(* CODESYS project SWDM240HES_S00107_20240509.project
   Company: ifm electronic
   Description: CR721S 2.25MByte Standard and Safety
   Title: ifmCR721S_TemplateProject
   Version: 3.1.4.1

Project tree, tasks and I/O mapping:
  StandardPLC : CR721S Standard, ifm electronic, order no. CR721S, version 3.1.4.1
    application Application
      libraries: ifmR360-3, * (ifm electronic); Standard, * (System); Util, * (System); SWMC_C_LIB, 3.5.15.7 (SW); CoDeSys External Library Template, 3.5.16.40 (3S - Smart Software Solutions GmbH); CoDeSys Common Library Template, 3.5.11.0 (3S - Smart Software Solutions GmbH)
      task Task (cyclic, interval t#10ms, priority 0) calls PLC_PRG
      IO_CONFIG/
        function block DiagFunction [FBD]
        program OUTPUT_CONFID [FBD]
        program ConfigDiagProt [FBD]
        program INPUT_CONFIG_PI [FBD]
        program INPUT_CONFIG [ST]
      EVC
      program PLC_PRG [FBD]
      CAN/
        program CAN1 [ST]
        program GPS_TONGXING_ALL [ST]
        program GPS_ALL [ST]
        program CanRecover [ST]
        program CAN0 [ST]
        program CAN2 [ST]
        program CAN_J [ST]
      data type FIFO_DUT
      SaveEngine/
        program SaveEngine [ST]
        global variables GVL_SaveEngine
        program SaveEngineControl [ST]
        program SaveEngineMode_1 [ST]
        program SaveEngineMode_2 [ST]
        program SaveEngineMode_3 [ST]
        program SaveEngineMode_4 [ST]
        program SaveEngineMode_5 [ST]
        program SaveEngineMode_6 [ST]
        program SaveEngineMode_7 [ST]
        program SaveEngineMode_8 [ST]
        program SaveEngineMode_19 [ST]
        program SaveEngineMode_10 [ST]
        program SaveEngineMode_11 [ST]
        program SaveEngineMode_12 [ST]
        program SaveEngineMode_9 [ST]
        program MainWinTension_Ave [ST]
        program Wt_Cal [ST]
      MOVE/
        program MastControl [ST]
        program worktime [ST]
        function block PID_JYF [ST]
        function block curve_quxian [ST]
        program control [ST]
        program inti_fasle [ST]
        program Joy_Analog_output [ST]
        function block ROTATE_AUTO [ST]
        function block MODE_ROTATE [ST]
      CAIJI/
        function block PRESSURE [ST]
        function block ANGLE_CAIJI_Y [ST]
        function block DEPTH [ST]
        function block Tension [ST]
        function block ZONGXIANJISUAN [ST]
        function block CAN_XY [FBD]
        function block censor_cali [FBD]
        function block FUEL_LEVEL [ST]
        function block ANGLE_CAIJI_X [ST]
        function block HYD_OIL_TEM [ST]
        program CAIJI_DEPTH [ST]
      GLV/
        global variables PersistentVars
        global variables Global_Variablen
        global variables IO_GLV
        global variables CAN_GVL
    HMI : HMI, ifm electronic, version 3.1.4.1
      User_LEDs : User_LEDs, ifm electronic, version 3.1.4.1
          input  UserLED0_I : LED_IEC_B_INPUT_MAPPING_TYPE  // UserLED0_I
          input  UserLED1_I : LED_IEC_B_INPUT_MAPPING_TYPE  // UserLED1_I
          input  UserLED2_I : LED_IEC_B_INPUT_MAPPING_TYPE  // UserLED2_I
          input  UserLED3_I : LED_IEC_B_INPUT_MAPPING_TYPE  // UserLED3_I
          output UserLED0_Q : LED_IEC_B_OUTPUT_MAPPING_TYPE  // User LED 0
          output UserLED1_Q : LED_IEC_B_OUTPUT_MAPPING_TYPE  // User LED 1
          output UserLED2_Q : LED_IEC_B_OUTPUT_MAPPING_TYPE  // User LED 2
          output UserLED3_Q : LED_IEC_B_OUTPUT_MAPPING_TYPE  // User LED 3
    Local_IO : Local_IO, ifm electronic, version 3.1.4.1
      System_Inputs : System_Inputs, ifm electronic, version 3.1.4.1
          input  VBB30 : IN_SYSTEM_VOLTAGE_INPUT_MAPPING_TYPE  // VBB30
          input  VBB15 : IN_SYSTEM_VOLTAGE_INPUT_MAPPING_TYPE  // VBB15
          input  TemperatureBoard0 : IN_TEMPERATURE_INPUT_MAPPING_TYPE  // TemperatureBoard0
          input  TemperatureChip0 : IN_TEMPERATURE_INPUT_MAPPING_TYPE  // TemperatureChip0
      Inputs : Inputs, ifm electronic, version 3.1.4.1
          input  IN0100_I : IN_MULTIFUNCTION_A_INPUT_MAPPING_TYPE  // IN0100_I
          input  IN0101_I : IN_MULTIFUNCTION_A_INPUT_MAPPING_TYPE  // IN0101_I
          input  IN0102_I : IN_MULTIFUNCTION_A_INPUT_MAPPING_TYPE  // IN0102_I
          input  IN0103_I : IN_MULTIFUNCTION_A_INPUT_MAPPING_TYPE  // IN0103_I
          input  IN0200_I : IN_MULTIFUNCTION_A_INPUT_MAPPING_TYPE  // IN0200_I
          input  IN0201_I : IN_MULTIFUNCTION_A_INPUT_MAPPING_TYPE  // IN0201_I
          input  IN0202_I : IN_MULTIFUNCTION_A_INPUT_MAPPING_TYPE  // IN0202_I
          input  IN0203_I : IN_MULTIFUNCTION_A_INPUT_MAPPING_TYPE  // IN0203_I
          input  IN0600_I : IN_MULTIFUNCTION_A_INPUT_MAPPING_TYPE  // IN0600_I
          input  IN0601_I : IN_MULTIFUNCTION_A_INPUT_MAPPING_TYPE  // IN0601_I
          input  IN0602_I : IN_MULTIFUNCTION_A_INPUT_MAPPING_TYPE  // IN0602_I
          input  IN0603_I : IN_MULTIFUNCTION_A_INPUT_MAPPING_TYPE  // IN0603_I
          input  IN0700_I : IN_MULTIFUNCTION_A_INPUT_MAPPING_TYPE  // IN0700_I
          input  IN0701_I : IN_MULTIFUNCTION_A_INPUT_MAPPING_TYPE  // IN0701_I
          input  IN0702_I : IN_MULTIFUNCTION_A_INPUT_MAPPING_TYPE  // IN0702_I
          input  IN0703_I : IN_MULTIFUNCTION_A_INPUT_MAPPING_TYPE  // IN0703_I
          input  IN1100_I : IN_MULTIFUNCTION_A_INPUT_MAPPING_TYPE  // IN1100_I
          input  IN1101_I : IN_MULTIFUNCTION_A_INPUT_MAPPING_TYPE  // IN1101_I
          input  IN1102_I : IN_MULTIFUNCTION_A_INPUT_MAPPING_TYPE  // IN1102_I
          input  IN1103_I : IN_MULTIFUNCTION_A_INPUT_MAPPING_TYPE  // IN1103_I
          input  IN1600_I : IN_MULTIFUNCTION_A_INPUT_MAPPING_TYPE  // IN1600_I
          input  IN1601_I : IN_MULTIFUNCTION_A_INPUT_MAPPING_TYPE  // IN1601_I
          input  IN1602_I : IN_MULTIFUNCTION_A_INPUT_MAPPING_TYPE  // IN1602_I
          input  IN1603_I : IN_MULTIFUNCTION_A_INPUT_MAPPING_TYPE  // IN1603_I
          input  IN0400_I : IN_RESISTOR_A_INPUT_MAPPING_TYPE  // IN0400_I
          input  IN0401_I : IN_RESISTOR_A_INPUT_MAPPING_TYPE  // IN0401_I
          input  IN0900_I : IN_RESISTOR_A_INPUT_MAPPING_TYPE  // IN0900_I
          input  IN0901_I : IN_RESISTOR_A_INPUT_MAPPING_TYPE  // IN0901_I
          input  IN1200_I : IN_DIGITAL_A_INPUT_MAPPING_TYPE  // IN1200_I
          input  IN1201_I : IN_DIGITAL_A_INPUT_MAPPING_TYPE  // IN1201_I
          input  IN1202_I : IN_DIGITAL_A_INPUT_MAPPING_TYPE  // IN1202_I
          input  IN1203_I : IN_DIGITAL_A_INPUT_MAPPING_TYPE  // IN1203_I
          input  IN1400_I : IN_DIGITAL_A_INPUT_MAPPING_TYPE  // IN1400_I
          input  IN1401_I : IN_DIGITAL_A_INPUT_MAPPING_TYPE  // IN1401_I
          input  IN1402_I : IN_DIGITAL_A_INPUT_MAPPING_TYPE  // IN1402_I
          input  IN1403_I : IN_DIGITAL_A_INPUT_MAPPING_TYPE  // IN1403_I
          input  IN1700_I : IN_DIGITAL_A_INPUT_MAPPING_TYPE  // IN1700_I
          input  IN1701_I : IN_DIGITAL_A_INPUT_MAPPING_TYPE  // IN1701_I
          input  IN1702_I : IN_DIGITAL_A_INPUT_MAPPING_TYPE  // IN1702_I
          input  IN1703_I : IN_DIGITAL_A_INPUT_MAPPING_TYPE  // IN1703_I
          input  IN1800_I : IN_DIGITAL_A_INPUT_MAPPING_TYPE  // IN1800_I
          input  IN1801_I : IN_DIGITAL_A_INPUT_MAPPING_TYPE  // IN1801_I
          input  IN1802_I : IN_DIGITAL_A_INPUT_MAPPING_TYPE  // IN1802_I
          input  IN1803_I : IN_DIGITAL_A_INPUT_MAPPING_TYPE  // IN1803_I
          input  IN0300_I : IN_DIGITAL_B_INPUT_MAPPING_TYPE  // IN0300_I
          input  IN0301_I : IN_DIGITAL_B_INPUT_MAPPING_TYPE  // IN0301_I
          input  IN0800_I : IN_DIGITAL_B_INPUT_MAPPING_TYPE  // IN0800_I
          input  IN0801_I : IN_DIGITAL_B_INPUT_MAPPING_TYPE  // IN0801_I
          input  IN1300_I : IN_DIGITAL_B_INPUT_MAPPING_TYPE  // IN1300_I
          input  IN1301_I : IN_DIGITAL_B_INPUT_MAPPING_TYPE  // IN1301_I
          input  IN1302_I : IN_DIGITAL_B_INPUT_MAPPING_TYPE  // IN1302_I
          input  IN1303_I : IN_DIGITAL_B_INPUT_MAPPING_TYPE  // IN1303_I
          input  COM_RESET_I : IN_COMMUNICATION_RESET_INPUT_MAPPING_TYPE  // COM_RESET_I
          input  IN0000_I : IN_FREQUENCY_B_CHANNEL_A_INPUT_MAPPING_TYPE  // IN0000_I
          input  IN0002_I : IN_FREQUENCY_B_CHANNEL_A_INPUT_MAPPING_TYPE  // IN0002_I
          input  IN0500_I : IN_FREQUENCY_B_CHANNEL_A_INPUT_MAPPING_TYPE  // IN0500_I
          input  IN0502_I : IN_FREQUENCY_B_CHANNEL_A_INPUT_MAPPING_TYPE  // IN0502_I
          input  IN1000_I : IN_FREQUENCY_B_CHANNEL_A_INPUT_MAPPING_TYPE  // IN1000_I
          input  IN1002_I : IN_FREQUENCY_B_CHANNEL_A_INPUT_MAPPING_TYPE  // IN1002_I
          input  IN1500_I : IN_FREQUENCY_B_CHANNEL_A_INPUT_MAPPING_TYPE  // IN1500_I
          input  IN1502_I : IN_FREQUENCY_B_CHANNEL_A_INPUT_MAPPING_TYPE  // IN1502_I
          input  IN0001_I : IN_FREQUENCY_B_CHANNEL_B_INPUT_MAPPING_TYPE  // IN0001_I
          input  IN0003_I : IN_FREQUENCY_B_CHANNEL_B_INPUT_MAPPING_TYPE  // IN0003_I
          input  IN0501_I : IN_FREQUENCY_B_CHANNEL_B_INPUT_MAPPING_TYPE  // IN0501_I
          input  IN0503_I : IN_FREQUENCY_B_CHANNEL_B_INPUT_MAPPING_TYPE  // IN0503_I
          input  IN1001_I : IN_FREQUENCY_B_CHANNEL_B_INPUT_MAPPING_TYPE  // IN1001_I
          input  IN1003_I : IN_FREQUENCY_B_CHANNEL_B_INPUT_MAPPING_TYPE  // IN1003_I
          input  IN1501_I : IN_FREQUENCY_B_CHANNEL_B_INPUT_MAPPING_TYPE  // IN1501_I
          input  IN1503_I : IN_FREQUENCY_B_CHANNEL_B_INPUT_MAPPING_TYPE  // IN1503_I
      Outputs : Outputs, ifm electronic, version 3.1.4.1
          input  OUT0006_I : OUT_PWM_40_BRIDGE_A_INPUT_MAPPING_TYPE  // OUT0006_I
          input  OUT0106_I : OUT_PWM_40_BRIDGE_A_INPUT_MAPPING_TYPE  // OUT0106_I
          input  OUT0206_I : OUT_PWM_40_BRIDGE_A_INPUT_MAPPING_TYPE  // OUT0206_I
          input  OUT0306_I : OUT_PWM_40_BRIDGE_A_INPUT_MAPPING_TYPE  // OUT0306_I
          input  OUT0406_I : OUT_PWM_40_BRIDGE_A_INPUT_MAPPING_TYPE  // OUT0406_I
          input  OUT0506_I : OUT_PWM_40_BRIDGE_A_INPUT_MAPPING_TYPE  // OUT0506_I
          input  OUT0008_I : OUT_PWM_40_A_INPUT_MAPPING_TYPE  // OUT0008_I
          input  OUT0108_I : OUT_PWM_40_A_INPUT_MAPPING_TYPE  // OUT0108_I
          input  OUT0208_I : OUT_PWM_40_A_INPUT_MAPPING_TYPE  // OUT0208_I
          input  OUT0308_I : OUT_PWM_40_A_INPUT_MAPPING_TYPE  // OUT0308_I
          input  OUT0408_I : OUT_PWM_40_A_INPUT_MAPPING_TYPE  // OUT0408_I
          input  OUT0508_I : OUT_PWM_40_A_INPUT_MAPPING_TYPE  // OUT0508_I
          input  OUT0000_I : OUT_PWM_25_A_INPUT_MAPPING_TYPE  // OUT0000_I
          input  OUT0002_I : OUT_PWM_25_A_INPUT_MAPPING_TYPE  // OUT0002_I
          input  OUT0004_I : OUT_PWM_25_A_INPUT_MAPPING_TYPE  // OUT0004_I
          input  OUT0100_I : OUT_PWM_25_A_INPUT_MAPPING_TYPE  // OUT0100_I
          input  OUT0102_I : OUT_PWM_25_A_INPUT_MAPPING_TYPE  // OUT0102_I
          input  OUT0104_I : OUT_PWM_25_A_INPUT_MAPPING_TYPE  // OUT0104_I
          input  OUT0200_I : OUT_PWM_25_A_INPUT_MAPPING_TYPE  // OUT0200_I
          input  OUT0202_I : OUT_PWM_25_A_INPUT_MAPPING_TYPE  // OUT0202_I
          input  OUT0204_I : OUT_PWM_25_A_INPUT_MAPPING_TYPE  // OUT0204_I
          input  OUT0300_I : OUT_PWM_25_A_INPUT_MAPPING_TYPE  // OUT0300_I
          input  OUT0302_I : OUT_PWM_25_A_INPUT_MAPPING_TYPE  // OUT0302_I
          input  OUT0304_I : OUT_PWM_25_A_INPUT_MAPPING_TYPE  // OUT0304_I
          input  OUT0400_I : OUT_PWM_25_A_INPUT_MAPPING_TYPE  // OUT0400_I
          input  OUT0402_I : OUT_PWM_25_A_INPUT_MAPPING_TYPE  // OUT0402_I
          input  OUT0404_I : OUT_PWM_25_A_INPUT_MAPPING_TYPE  // OUT0404_I
          input  OUT0500_I : OUT_PWM_25_A_INPUT_MAPPING_TYPE  // OUT0500_I
          input  OUT0502_I : OUT_PWM_25_A_INPUT_MAPPING_TYPE  // OUT0502_I
          input  OUT0504_I : OUT_PWM_25_A_INPUT_MAPPING_TYPE  // OUT0504_I
          input  OUT3001_I : OUT_VOLTAGE_A_INPUT_MAPPING_TYPE  // OUT3001_I
          input  OUT3002_I : OUT_VOLTAGE_A_INPUT_MAPPING_TYPE  // OUT3002_I
          input  OUT3000_I : OUT_SUPPLY_A_INPUT_MAPPING_TYPE  // OUT3000_I
          input  OUT0001_I : OUT_PWM_25_B_INPUT_MAPPING_TYPE  // OUT0001_I
          input  OUT0003_I : OUT_PWM_25_B_INPUT_MAPPING_TYPE  // OUT0003_I
          input  OUT0005_I : OUT_PWM_25_B_INPUT_MAPPING_TYPE  // OUT0005_I
          input  OUT0101_I : OUT_PWM_25_B_INPUT_MAPPING_TYPE  // OUT0101_I
          input  OUT0103_I : OUT_PWM_25_B_INPUT_MAPPING_TYPE  // OUT0103_I
          input  OUT0105_I : OUT_PWM_25_B_INPUT_MAPPING_TYPE  // OUT0105_I
          input  OUT0201_I : OUT_PWM_25_B_INPUT_MAPPING_TYPE  // OUT0201_I
          input  OUT0203_I : OUT_PWM_25_B_INPUT_MAPPING_TYPE  // OUT0203_I
          input  OUT0205_I : OUT_PWM_25_B_INPUT_MAPPING_TYPE  // OUT0205_I
          input  OUT0301_I : OUT_PWM_25_B_INPUT_MAPPING_TYPE  // OUT0301_I
          input  OUT0303_I : OUT_PWM_25_B_INPUT_MAPPING_TYPE  // OUT0303_I
          input  OUT0305_I : OUT_PWM_25_B_INPUT_MAPPING_TYPE  // OUT0305_I
          input  OUT0401_I : OUT_PWM_25_B_INPUT_MAPPING_TYPE  // OUT0401_I
          input  OUT0403_I : OUT_PWM_25_B_INPUT_MAPPING_TYPE  // OUT0403_I
          input  OUT0405_I : OUT_PWM_25_B_INPUT_MAPPING_TYPE  // OUT0405_I
          input  OUT0501_I : OUT_PWM_25_B_INPUT_MAPPING_TYPE  // OUT0501_I
          input  OUT0503_I : OUT_PWM_25_B_INPUT_MAPPING_TYPE  // OUT0503_I
          input  OUT0505_I : OUT_PWM_25_B_INPUT_MAPPING_TYPE  // OUT0505_I
          input  OUT0007_I : OUT_PWM_40_BRIDGE_A_INPUT_MAPPING_TYPE  // OUT0007_I
          input  OUT0107_I : OUT_PWM_40_BRIDGE_A_INPUT_MAPPING_TYPE  // OUT0107_I
          input  OUT0207_I : OUT_PWM_40_BRIDGE_A_INPUT_MAPPING_TYPE  // OUT0207_I
          input  OUT0307_I : OUT_PWM_40_BRIDGE_A_INPUT_MAPPING_TYPE  // OUT0307_I
          input  OUT0407_I : OUT_PWM_40_BRIDGE_A_INPUT_MAPPING_TYPE  // OUT0407_I
          input  OUT0507_I : OUT_PWM_40_BRIDGE_A_INPUT_MAPPING_TYPE  // OUT0507_I
          output OUT0006_Q : OUT_PWM_40_BRIDGE_A_OUTPUT_MAPPING_TYPE  // OUT0006_Q
          output OUT0106_Q : OUT_PWM_40_BRIDGE_A_OUTPUT_MAPPING_TYPE  // OUT0106_Q
          output OUT0206_Q : OUT_PWM_40_BRIDGE_A_OUTPUT_MAPPING_TYPE  // OUT0206_Q
          output OUT0306_Q : OUT_PWM_40_BRIDGE_A_OUTPUT_MAPPING_TYPE  // OUT0306_Q
          output OUT0406_Q : OUT_PWM_40_BRIDGE_A_OUTPUT_MAPPING_TYPE  // OUT0406_Q
          output OUT0506_Q : OUT_PWM_40_BRIDGE_A_OUTPUT_MAPPING_TYPE  // OUT0506_Q
          output OUT0008_Q : OUT_PWM_40_A_OUTPUT_MAPPING_TYPE  // OUT0008_Q
          output OUT0108_Q : OUT_PWM_40_A_OUTPUT_MAPPING_TYPE  // OUT0108_Q
          output OUT0208_Q : OUT_PWM_40_A_OUTPUT_MAPPING_TYPE  // OUT0208_Q
          output OUT0308_Q : OUT_PWM_40_A_OUTPUT_MAPPING_TYPE  // OUT0308_Q
          output OUT0408_Q : OUT_PWM_40_A_OUTPUT_MAPPING_TYPE  // OUT0408_Q
          output OUT0508_Q : OUT_PWM_40_A_OUTPUT_MAPPING_TYPE  // OUT0508_Q
          output OUT0000_Q : OUT_PWM_25_A_OUTPUT_MAPPING_TYPE  // OUT0000_Q
          output OUT0002_Q : OUT_PWM_25_A_OUTPUT_MAPPING_TYPE  // OUT0002_Q
          output OUT0004_Q : OUT_PWM_25_A_OUTPUT_MAPPING_TYPE  // OUT0004_Q
          output OUT0100_Q : OUT_PWM_25_A_OUTPUT_MAPPING_TYPE  // OUT0100_Q
          output OUT0102_Q : OUT_PWM_25_A_OUTPUT_MAPPING_TYPE  // OUT0102_Q
          output OUT0104_Q : OUT_PWM_25_A_OUTPUT_MAPPING_TYPE  // OUT0104_Q
          output OUT0200_Q : OUT_PWM_25_A_OUTPUT_MAPPING_TYPE  // OUT0200_Q
          output OUT0202_Q : OUT_PWM_25_A_OUTPUT_MAPPING_TYPE  // OUT0202_Q
          output OUT0204_Q : OUT_PWM_25_A_OUTPUT_MAPPING_TYPE  // OUT0204_Q
          output OUT0300_Q : OUT_PWM_25_A_OUTPUT_MAPPING_TYPE  // OUT0300_Q
          output OUT0302_Q : OUT_PWM_25_A_OUTPUT_MAPPING_TYPE  // OUT0302_Q
          output OUT0304_Q : OUT_PWM_25_A_OUTPUT_MAPPING_TYPE  // OUT0304_Q
          output OUT0400_Q : OUT_PWM_25_A_OUTPUT_MAPPING_TYPE  // OUT0400_Q
          output OUT0402_Q : OUT_PWM_25_A_OUTPUT_MAPPING_TYPE  // OUT0402_Q
          output OUT0404_Q : OUT_PWM_25_A_OUTPUT_MAPPING_TYPE  // OUT0404_Q
          output OUT0500_Q : OUT_PWM_25_A_OUTPUT_MAPPING_TYPE  // OUT0500_Q
          output OUT0502_Q : OUT_PWM_25_A_OUTPUT_MAPPING_TYPE  // OUT0502_Q
          output OUT0504_Q : OUT_PWM_25_A_OUTPUT_MAPPING_TYPE  // OUT0504_Q
          output OUT3001_Q : OUT_VOLTAGE_A_OUTPUT_MAPPING_TYPE  // OUT3001_Q
          output OUT3002_Q : OUT_VOLTAGE_A_OUTPUT_MAPPING_TYPE  // OUT3002_Q
          output OUT3000_Q : OUT_SUPPLY_A_OUTPUT_MAPPING_TYPE  // OUT3000_Q
          output OUT0001_Q : OUT_PWM_25_B_OUTPUT_MAPPING_TYPE  // OUT0001_Q
          output OUT0003_Q : OUT_PWM_25_B_OUTPUT_MAPPING_TYPE  // OUT0003_Q
          output OUT0005_Q : OUT_PWM_25_B_OUTPUT_MAPPING_TYPE  // OUT0005_Q
          output OUT0101_Q : OUT_PWM_25_B_OUTPUT_MAPPING_TYPE  // OUT0101_Q
          output OUT0103_Q : OUT_PWM_25_B_OUTPUT_MAPPING_TYPE  // OUT0103_Q
          output OUT0105_Q : OUT_PWM_25_B_OUTPUT_MAPPING_TYPE  // OUT0105_Q
          output OUT0201_Q : OUT_PWM_25_B_OUTPUT_MAPPING_TYPE  // OUT0201_Q
          output OUT0203_Q : OUT_PWM_25_B_OUTPUT_MAPPING_TYPE  // OUT0203_Q
          output OUT0205_Q : OUT_PWM_25_B_OUTPUT_MAPPING_TYPE  // OUT0205_Q
          output OUT0301_Q : OUT_PWM_25_B_OUTPUT_MAPPING_TYPE  // OUT0301_Q
          output OUT0303_Q : OUT_PWM_25_B_OUTPUT_MAPPING_TYPE  // OUT0303_Q
          output OUT0305_Q : OUT_PWM_25_B_OUTPUT_MAPPING_TYPE  // OUT0305_Q
          output OUT0401_Q : OUT_PWM_25_B_OUTPUT_MAPPING_TYPE  // OUT0401_Q
          output OUT0403_Q : OUT_PWM_25_B_OUTPUT_MAPPING_TYPE  // OUT0403_Q
          output OUT0405_Q : OUT_PWM_25_B_OUTPUT_MAPPING_TYPE  // OUT0405_Q
          output OUT0501_Q : OUT_PWM_25_B_OUTPUT_MAPPING_TYPE  // OUT0501_Q
          output OUT0503_Q : OUT_PWM_25_B_OUTPUT_MAPPING_TYPE  // OUT0503_Q
          output OUT0505_Q : OUT_PWM_25_B_OUTPUT_MAPPING_TYPE  // OUT0505_Q
          output OUT0007_Q : OUT_PWM_40_BRIDGE_A_OUTPUT_MAPPING_TYPE  // OUT0007_Q
          output OUT0107_Q : OUT_PWM_40_BRIDGE_A_OUTPUT_MAPPING_TYPE  // OUT0107_Q
          output OUT0207_Q : OUT_PWM_40_BRIDGE_A_OUTPUT_MAPPING_TYPE  // OUT0207_Q
          output OUT0307_Q : OUT_PWM_40_BRIDGE_A_OUTPUT_MAPPING_TYPE  // OUT0307_Q
          output OUT0407_Q : OUT_PWM_40_BRIDGE_A_OUTPUT_MAPPING_TYPE  // OUT0407_Q
          output OUT0507_Q : OUT_PWM_40_BRIDGE_A_OUTPUT_MAPPING_TYPE  // OUT0507_Q
      System_Outputs : System_Outputs, ifm electronic, version 3.1.4.1
          input  VBB0_SW_I : OUT_GROUP_SWITCH_INPUT_MAPPING_TYPE  // VBB0_SW_I
          input  VBB1_SW_I : OUT_GROUP_SWITCH_INPUT_MAPPING_TYPE  // VBB1_SW_I
          input  VBB2_SW_I : OUT_GROUP_SWITCH_INPUT_MAPPING_TYPE  // VBB2_SW_I
          input  VBB3_SW_I : OUT_GROUP_SWITCH_INPUT_MAPPING_TYPE  // VBB3_SW_I
          input  VBB4_SW_I : OUT_GROUP_SWITCH_INPUT_MAPPING_TYPE  // VBB4_SW_I
          input  VBB5_SW_I : OUT_GROUP_SWITCH_INPUT_MAPPING_TYPE  // VBB5_SW_I
          output VBB0_SW_Q : OUT_GROUP_SWITCH_OUTPUT_MAPPING_TYPE  // VBB0_SW_Q
          output VBB1_SW_Q : OUT_GROUP_SWITCH_OUTPUT_MAPPING_TYPE  // VBB1_SW_Q
          output VBB2_SW_Q : OUT_GROUP_SWITCH_OUTPUT_MAPPING_TYPE  // VBB2_SW_Q
          output VBB3_SW_Q : OUT_GROUP_SWITCH_OUTPUT_MAPPING_TYPE  // VBB3_SW_Q
          output VBB4_SW_Q : OUT_GROUP_SWITCH_OUTPUT_MAPPING_TYPE  // VBB4_SW_Q
          output VBB5_SW_Q : OUT_GROUP_SWITCH_OUTPUT_MAPPING_TYPE  // VBB5_SW_Q
          output SUPPLY_SWITCH_Q : OUT_SYS_SWITCH_OUTPUT_MAPPING_TYPE  // SUPPLY_SWITCH_Q
    Communication : Communication, ifm electronic, version 3.1.4.1
      CAN : CAN, ifm electronic, version 3.1.4.1
        CANbus_0 : CANbus, ifm electronic, version 1.0.1.1
      Ethernet : Ethernet, ifm electronic, version 3.1.4.1
  SafetyPLC : CR721S SIL2, ifm electronic, order no. CR721S, version 3.1.4.1
    application Application
      libraries: ifmR360-3, * (ifm electronic); Standard, * (System); Util, * (System)
      global variables EVL
    HMI : HMI, ifm electronic, version 3.1.4.1
      User_LEDs : User_LEDs, ifm electronic, version 3.1.4.1
          input  UserLED0_I : LED_IEC_B_INPUT_MAPPING_TYPE  // UserLED0_I
          input  UserLED1_I : LED_IEC_B_INPUT_MAPPING_TYPE  // UserLED1_I
          input  UserLED2_I : LED_IEC_B_INPUT_MAPPING_TYPE  // UserLED2_I
          input  UserLED3_I : LED_IEC_B_INPUT_MAPPING_TYPE  // UserLED3_I
          output UserLED0_Q : LED_IEC_B_OUTPUT_MAPPING_TYPE  // User LED 0
          output UserLED1_Q : LED_IEC_B_OUTPUT_MAPPING_TYPE  // User LED 1
          output UserLED2_Q : LED_IEC_B_OUTPUT_MAPPING_TYPE  // User LED 2
          output UserLED3_Q : LED_IEC_B_OUTPUT_MAPPING_TYPE  // User LED 3
    Local_IO : Local_IO, ifm electronic, version 3.1.4.1
      System_Outputs : System_Outputs, ifm electronic, version 3.1.4.1
          input  VBB0_SW_I : OUT_GROUP_SWITCH_INPUT_MAPPING_TYPE  // VBB0_SW_I
          input  VBB1_SW_I : OUT_GROUP_SWITCH_INPUT_MAPPING_TYPE  // VBB1_SW_I
          input  VBB2_SW_I : OUT_GROUP_SWITCH_INPUT_MAPPING_TYPE  // VBB2_SW_I
          input  VBB3_SW_I : OUT_GROUP_SWITCH_INPUT_MAPPING_TYPE  // VBB3_SW_I
          input  VBB4_SW_I : OUT_GROUP_SWITCH_INPUT_MAPPING_TYPE  // VBB4_SW_I
          input  VBB5_SW_I : OUT_GROUP_SWITCH_INPUT_MAPPING_TYPE  // VBB5_SW_I
          output VBB0_SW_Q : OUT_GROUP_SWITCH_OUTPUT_MAPPING_TYPE  // VBB0_SW_Q
          output VBB1_SW_Q : OUT_GROUP_SWITCH_OUTPUT_MAPPING_TYPE  // VBB1_SW_Q
          output VBB2_SW_Q : OUT_GROUP_SWITCH_OUTPUT_MAPPING_TYPE  // VBB2_SW_Q
          output VBB3_SW_Q : OUT_GROUP_SWITCH_OUTPUT_MAPPING_TYPE  // VBB3_SW_Q
          output VBB4_SW_Q : OUT_GROUP_SWITCH_OUTPUT_MAPPING_TYPE  // VBB4_SW_Q
          output VBB5_SW_Q : OUT_GROUP_SWITCH_OUTPUT_MAPPING_TYPE  // VBB5_SW_Q
          output SUPPLY_SWITCH_Q : OUT_SYS_SWITCH_OUTPUT_MAPPING_TYPE  // SUPPLY_SWITCH_Q
      Outputs : Outputs, ifm electronic, version 3.1.4.1
          input  OUT0006_I : OUT_PWM_40_BRIDGE_A_INPUT_MAPPING_TYPE  // OUT0006_I
          input  OUT0106_I : OUT_PWM_40_BRIDGE_A_INPUT_MAPPING_TYPE  // OUT0106_I
          input  OUT0206_I : OUT_PWM_40_BRIDGE_A_INPUT_MAPPING_TYPE  // OUT0206_I
          input  OUT0306_I : OUT_PWM_40_BRIDGE_A_INPUT_MAPPING_TYPE  // OUT0306_I
          input  OUT0406_I : OUT_PWM_40_BRIDGE_A_INPUT_MAPPING_TYPE  // OUT0406_I
          input  OUT0506_I : OUT_PWM_40_BRIDGE_A_INPUT_MAPPING_TYPE  // OUT0506_I
          input  OUT0008_I : OUT_PWM_40_A_INPUT_MAPPING_TYPE  // OUT0008_I
          input  OUT0108_I : OUT_PWM_40_A_INPUT_MAPPING_TYPE  // OUT0108_I
          input  OUT0208_I : OUT_PWM_40_A_INPUT_MAPPING_TYPE  // OUT0208_I
          input  OUT0308_I : OUT_PWM_40_A_INPUT_MAPPING_TYPE  // OUT0308_I
          input  OUT0408_I : OUT_PWM_40_A_INPUT_MAPPING_TYPE  // OUT0408_I
          input  OUT0508_I : OUT_PWM_40_A_INPUT_MAPPING_TYPE  // OUT0508_I
          input  OUT0000_I : OUT_PWM_25_A_INPUT_MAPPING_TYPE  // OUT0000_I
          input  OUT0002_I : OUT_PWM_25_A_INPUT_MAPPING_TYPE  // OUT0002_I
          input  OUT0004_I : OUT_PWM_25_A_INPUT_MAPPING_TYPE  // OUT0004_I
          input  OUT0100_I : OUT_PWM_25_A_INPUT_MAPPING_TYPE  // OUT0100_I
          input  OUT0102_I : OUT_PWM_25_A_INPUT_MAPPING_TYPE  // OUT0102_I
          input  OUT0104_I : OUT_PWM_25_A_INPUT_MAPPING_TYPE  // OUT0104_I
          input  OUT0200_I : OUT_PWM_25_A_INPUT_MAPPING_TYPE  // OUT0200_I
          input  OUT0202_I : OUT_PWM_25_A_INPUT_MAPPING_TYPE  // OUT0202_I
          input  OUT0204_I : OUT_PWM_25_A_INPUT_MAPPING_TYPE  // OUT0204_I
          input  OUT0300_I : OUT_PWM_25_A_INPUT_MAPPING_TYPE  // OUT0300_I
          input  OUT0302_I : OUT_PWM_25_A_INPUT_MAPPING_TYPE  // OUT0302_I
          input  OUT0304_I : OUT_PWM_25_A_INPUT_MAPPING_TYPE  // OUT0304_I
          input  OUT0400_I : OUT_PWM_25_A_INPUT_MAPPING_TYPE  // OUT0400_I
          input  OUT0402_I : OUT_PWM_25_A_INPUT_MAPPING_TYPE  // OUT0402_I
          input  OUT0404_I : OUT_PWM_25_A_INPUT_MAPPING_TYPE  // OUT0404_I
          input  OUT0500_I : OUT_PWM_25_A_INPUT_MAPPING_TYPE  // OUT0500_I
          input  OUT0502_I : OUT_PWM_25_A_INPUT_MAPPING_TYPE  // OUT0502_I
          input  OUT0504_I : OUT_PWM_25_A_INPUT_MAPPING_TYPE  // OUT0504_I
          input  OUT3001_I : OUT_VOLTAGE_A_INPUT_MAPPING_TYPE  // OUT3001_I
          input  OUT3002_I : OUT_VOLTAGE_A_INPUT_MAPPING_TYPE  // OUT3002_I
          input  OUT3000_I : OUT_SUPPLY_A_INPUT_MAPPING_TYPE  // OUT3000_I
          input  OUT0001_I : OUT_PWM_25_B_INPUT_MAPPING_TYPE  // OUT0001_I
          input  OUT0003_I : OUT_PWM_25_B_INPUT_MAPPING_TYPE  // OUT0003_I
          input  OUT0005_I : OUT_PWM_25_B_INPUT_MAPPING_TYPE  // OUT0005_I
          input  OUT0101_I : OUT_PWM_25_B_INPUT_MAPPING_TYPE  // OUT0101_I
          input  OUT0103_I : OUT_PWM_25_B_INPUT_MAPPING_TYPE  // OUT0103_I
          input  OUT0105_I : OUT_PWM_25_B_INPUT_MAPPING_TYPE  // OUT0105_I
          input  OUT0201_I : OUT_PWM_25_B_INPUT_MAPPING_TYPE  // OUT0201_I
          input  OUT0203_I : OUT_PWM_25_B_INPUT_MAPPING_TYPE  // OUT0203_I
          input  OUT0205_I : OUT_PWM_25_B_INPUT_MAPPING_TYPE  // OUT0205_I
          input  OUT0301_I : OUT_PWM_25_B_INPUT_MAPPING_TYPE  // OUT0301_I
          input  OUT0303_I : OUT_PWM_25_B_INPUT_MAPPING_TYPE  // OUT0303_I
          input  OUT0305_I : OUT_PWM_25_B_INPUT_MAPPING_TYPE  // OUT0305_I
          input  OUT0401_I : OUT_PWM_25_B_INPUT_MAPPING_TYPE  // OUT0401_I
          input  OUT0403_I : OUT_PWM_25_B_INPUT_MAPPING_TYPE  // OUT0403_I
          input  OUT0405_I : OUT_PWM_25_B_INPUT_MAPPING_TYPE  // OUT0405_I
          input  OUT0501_I : OUT_PWM_25_B_INPUT_MAPPING_TYPE  // OUT0501_I
          input  OUT0503_I : OUT_PWM_25_B_INPUT_MAPPING_TYPE  // OUT0503_I
          input  OUT0505_I : OUT_PWM_25_B_INPUT_MAPPING_TYPE  // OUT0505_I
          input  OUT0007_I : OUT_PWM_40_BRIDGE_A_INPUT_MAPPING_TYPE  // OUT0007_I
          input  OUT0107_I : OUT_PWM_40_BRIDGE_A_INPUT_MAPPING_TYPE  // OUT0107_I
          input  OUT0207_I : OUT_PWM_40_BRIDGE_A_INPUT_MAPPING_TYPE  // OUT0207_I
          input  OUT0307_I : OUT_PWM_40_BRIDGE_A_INPUT_MAPPING_TYPE  // OUT0307_I
          input  OUT0407_I : OUT_PWM_40_BRIDGE_A_INPUT_MAPPING_TYPE  // OUT0407_I
          input  OUT0507_I : OUT_PWM_40_BRIDGE_A_INPUT_MAPPING_TYPE  // OUT0507_I
          output OUT0006_Q : OUT_PWM_40_BRIDGE_A_OUTPUT_MAPPING_TYPE  // OUT0006_Q
          output OUT0106_Q : OUT_PWM_40_BRIDGE_A_OUTPUT_MAPPING_TYPE  // OUT0106_Q
          output OUT0206_Q : OUT_PWM_40_BRIDGE_A_OUTPUT_MAPPING_TYPE  // OUT0206_Q
          output OUT0306_Q : OUT_PWM_40_BRIDGE_A_OUTPUT_MAPPING_TYPE  // OUT0306_Q
          output OUT0406_Q : OUT_PWM_40_BRIDGE_A_OUTPUT_MAPPING_TYPE  // OUT0406_Q
          output OUT0506_Q : OUT_PWM_40_BRIDGE_A_OUTPUT_MAPPING_TYPE  // OUT0506_Q
          output OUT0008_Q : OUT_PWM_40_A_OUTPUT_MAPPING_TYPE  // OUT0008_Q
          output OUT0108_Q : OUT_PWM_40_A_OUTPUT_MAPPING_TYPE  // OUT0108_Q
          output OUT0208_Q : OUT_PWM_40_A_OUTPUT_MAPPING_TYPE  // OUT0208_Q
          output OUT0308_Q : OUT_PWM_40_A_OUTPUT_MAPPING_TYPE  // OUT0308_Q
          output OUT0408_Q : OUT_PWM_40_A_OUTPUT_MAPPING_TYPE  // OUT0408_Q
          output OUT0508_Q : OUT_PWM_40_A_OUTPUT_MAPPING_TYPE  // OUT0508_Q
          output OUT0000_Q : OUT_PWM_25_A_OUTPUT_MAPPING_TYPE  // OUT0000_Q
          output OUT0002_Q : OUT_PWM_25_A_OUTPUT_MAPPING_TYPE  // OUT0002_Q
          output OUT0004_Q : OUT_PWM_25_A_OUTPUT_MAPPING_TYPE  // OUT0004_Q
          output OUT0100_Q : OUT_PWM_25_A_OUTPUT_MAPPING_TYPE  // OUT0100_Q
          output OUT0102_Q : OUT_PWM_25_A_OUTPUT_MAPPING_TYPE  // OUT0102_Q
          output OUT0104_Q : OUT_PWM_25_A_OUTPUT_MAPPING_TYPE  // OUT0104_Q
          output OUT0200_Q : OUT_PWM_25_A_OUTPUT_MAPPING_TYPE  // OUT0200_Q
          output OUT0202_Q : OUT_PWM_25_A_OUTPUT_MAPPING_TYPE  // OUT0202_Q
          output OUT0204_Q : OUT_PWM_25_A_OUTPUT_MAPPING_TYPE  // OUT0204_Q
          output OUT0300_Q : OUT_PWM_25_A_OUTPUT_MAPPING_TYPE  // OUT0300_Q
          output OUT0302_Q : OUT_PWM_25_A_OUTPUT_MAPPING_TYPE  // OUT0302_Q
          output OUT0304_Q : OUT_PWM_25_A_OUTPUT_MAPPING_TYPE  // OUT0304_Q
          output OUT0400_Q : OUT_PWM_25_A_OUTPUT_MAPPING_TYPE  // OUT0400_Q
          output OUT0402_Q : OUT_PWM_25_A_OUTPUT_MAPPING_TYPE  // OUT0402_Q
          output OUT0404_Q : OUT_PWM_25_A_OUTPUT_MAPPING_TYPE  // OUT0404_Q
          output OUT0500_Q : OUT_PWM_25_A_OUTPUT_MAPPING_TYPE  // OUT0500_Q
          output OUT0502_Q : OUT_PWM_25_A_OUTPUT_MAPPING_TYPE  // OUT0502_Q
          output OUT0504_Q : OUT_PWM_25_A_OUTPUT_MAPPING_TYPE  // OUT0504_Q
          output OUT3001_Q : OUT_VOLTAGE_A_OUTPUT_MAPPING_TYPE  // OUT3001_Q
          output OUT3002_Q : OUT_VOLTAGE_A_OUTPUT_MAPPING_TYPE  // OUT3002_Q
          output OUT3000_Q : OUT_SUPPLY_A_OUTPUT_MAPPING_TYPE  // OUT3000_Q
          output OUT0001_Q : OUT_PWM_25_B_OUTPUT_MAPPING_TYPE  // OUT0001_Q
          output OUT0003_Q : OUT_PWM_25_B_OUTPUT_MAPPING_TYPE  // OUT0003_Q
          output OUT0005_Q : OUT_PWM_25_B_OUTPUT_MAPPING_TYPE  // OUT0005_Q
          output OUT0101_Q : OUT_PWM_25_B_OUTPUT_MAPPING_TYPE  // OUT0101_Q
          output OUT0103_Q : OUT_PWM_25_B_OUTPUT_MAPPING_TYPE  // OUT0103_Q
          output OUT0105_Q : OUT_PWM_25_B_OUTPUT_MAPPING_TYPE  // OUT0105_Q
          output OUT0201_Q : OUT_PWM_25_B_OUTPUT_MAPPING_TYPE  // OUT0201_Q
          output OUT0203_Q : OUT_PWM_25_B_OUTPUT_MAPPING_TYPE  // OUT0203_Q
          output OUT0205_Q : OUT_PWM_25_B_OUTPUT_MAPPING_TYPE  // OUT0205_Q
          output OUT0301_Q : OUT_PWM_25_B_OUTPUT_MAPPING_TYPE  // OUT0301_Q
          output OUT0303_Q : OUT_PWM_25_B_OUTPUT_MAPPING_TYPE  // OUT0303_Q
          output OUT0305_Q : OUT_PWM_25_B_OUTPUT_MAPPING_TYPE  // OUT0305_Q
          output OUT0401_Q : OUT_PWM_25_B_OUTPUT_MAPPING_TYPE  // OUT0401_Q
          output OUT0403_Q : OUT_PWM_25_B_OUTPUT_MAPPING_TYPE  // OUT0403_Q
          output OUT0405_Q : OUT_PWM_25_B_OUTPUT_MAPPING_TYPE  // OUT0405_Q
          output OUT0501_Q : OUT_PWM_25_B_OUTPUT_MAPPING_TYPE  // OUT0501_Q
          output OUT0503_Q : OUT_PWM_25_B_OUTPUT_MAPPING_TYPE  // OUT0503_Q
          output OUT0505_Q : OUT_PWM_25_B_OUTPUT_MAPPING_TYPE  // OUT0505_Q
          output OUT0007_Q : OUT_PWM_40_BRIDGE_A_OUTPUT_MAPPING_TYPE  // OUT0007_Q
          output OUT0107_Q : OUT_PWM_40_BRIDGE_A_OUTPUT_MAPPING_TYPE  // OUT0107_Q
          output OUT0207_Q : OUT_PWM_40_BRIDGE_A_OUTPUT_MAPPING_TYPE  // OUT0207_Q
          output OUT0307_Q : OUT_PWM_40_BRIDGE_A_OUTPUT_MAPPING_TYPE  // OUT0307_Q
          output OUT0407_Q : OUT_PWM_40_BRIDGE_A_OUTPUT_MAPPING_TYPE  // OUT0407_Q
          output OUT0507_Q : OUT_PWM_40_BRIDGE_A_OUTPUT_MAPPING_TYPE  // OUT0507_Q
      System_Inputs : System_Inputs, ifm electronic, version 3.1.4.1
          input  VBB30 : IN_SYSTEM_VOLTAGE_INPUT_MAPPING_TYPE  // VBB30
          input  VBB15 : IN_SYSTEM_VOLTAGE_INPUT_MAPPING_TYPE  // VBB15
          input  TemperatureBoard0 : IN_TEMPERATURE_INPUT_MAPPING_TYPE  // TemperatureBoard0
          input  TemperatureChip0 : IN_TEMPERATURE_INPUT_MAPPING_TYPE  // TemperatureChip0
      Inputs : Inputs, ifm electronic, version 3.1.4.1
          input  IN0100_I : IN_MULTIFUNCTION_A_INPUT_MAPPING_TYPE  // IN0100_I
          input  IN0101_I : IN_MULTIFUNCTION_A_INPUT_MAPPING_TYPE  // IN0101_I
          input  IN0102_I : IN_MULTIFUNCTION_A_INPUT_MAPPING_TYPE  // IN0102_I
          input  IN0103_I : IN_MULTIFUNCTION_A_INPUT_MAPPING_TYPE  // IN0103_I
          input  IN0200_I : IN_MULTIFUNCTION_A_INPUT_MAPPING_TYPE  // IN0200_I
          input  IN0201_I : IN_MULTIFUNCTION_A_INPUT_MAPPING_TYPE  // IN0201_I
          input  IN0202_I : IN_MULTIFUNCTION_A_INPUT_MAPPING_TYPE  // IN0202_I
          input  IN0203_I : IN_MULTIFUNCTION_A_INPUT_MAPPING_TYPE  // IN0203_I
          input  IN0600_I : IN_MULTIFUNCTION_A_INPUT_MAPPING_TYPE  // IN0600_I
          input  IN0601_I : IN_MULTIFUNCTION_A_INPUT_MAPPING_TYPE  // IN0601_I
          input  IN0602_I : IN_MULTIFUNCTION_A_INPUT_MAPPING_TYPE  // IN0602_I
          input  IN0603_I : IN_MULTIFUNCTION_A_INPUT_MAPPING_TYPE  // IN0603_I
          input  IN0700_I : IN_MULTIFUNCTION_A_INPUT_MAPPING_TYPE  // IN0700_I
          input  IN0701_I : IN_MULTIFUNCTION_A_INPUT_MAPPING_TYPE  // IN0701_I
          input  IN0702_I : IN_MULTIFUNCTION_A_INPUT_MAPPING_TYPE  // IN0702_I
          input  IN0703_I : IN_MULTIFUNCTION_A_INPUT_MAPPING_TYPE  // IN0703_I
          input  IN1100_I : IN_MULTIFUNCTION_A_INPUT_MAPPING_TYPE  // IN1100_I
          input  IN1101_I : IN_MULTIFUNCTION_A_INPUT_MAPPING_TYPE  // IN1101_I
          input  IN1102_I : IN_MULTIFUNCTION_A_INPUT_MAPPING_TYPE  // IN1102_I
          input  IN1103_I : IN_MULTIFUNCTION_A_INPUT_MAPPING_TYPE  // IN1103_I
          input  IN1600_I : IN_MULTIFUNCTION_A_INPUT_MAPPING_TYPE  // IN1600_I
          input  IN1601_I : IN_MULTIFUNCTION_A_INPUT_MAPPING_TYPE  // IN1601_I
          input  IN1602_I : IN_MULTIFUNCTION_A_INPUT_MAPPING_TYPE  // IN1602_I
          input  IN1603_I : IN_MULTIFUNCTION_A_INPUT_MAPPING_TYPE  // IN1603_I
          input  IN0400_I : IN_RESISTOR_A_INPUT_MAPPING_TYPE  // IN0400_I
          input  IN0401_I : IN_RESISTOR_A_INPUT_MAPPING_TYPE  // IN0401_I
          input  IN0900_I : IN_RESISTOR_A_INPUT_MAPPING_TYPE  // IN0900_I
          input  IN0901_I : IN_RESISTOR_A_INPUT_MAPPING_TYPE  // IN0901_I
          input  IN1200_I : IN_DIGITAL_A_INPUT_MAPPING_TYPE  // IN1200_I
          input  IN1201_I : IN_DIGITAL_A_INPUT_MAPPING_TYPE  // IN1201_I
          input  IN1202_I : IN_DIGITAL_A_INPUT_MAPPING_TYPE  // IN1202_I
          input  IN1203_I : IN_DIGITAL_A_INPUT_MAPPING_TYPE  // IN1203_I
          input  IN1400_I : IN_DIGITAL_A_INPUT_MAPPING_TYPE  // IN1400_I
          input  IN1401_I : IN_DIGITAL_A_INPUT_MAPPING_TYPE  // IN1401_I
          input  IN1402_I : IN_DIGITAL_A_INPUT_MAPPING_TYPE  // IN1402_I
          input  IN1403_I : IN_DIGITAL_A_INPUT_MAPPING_TYPE  // IN1403_I
          input  IN1700_I : IN_DIGITAL_A_INPUT_MAPPING_TYPE  // IN1700_I
          input  IN1701_I : IN_DIGITAL_A_INPUT_MAPPING_TYPE  // IN1701_I
          input  IN1702_I : IN_DIGITAL_A_INPUT_MAPPING_TYPE  // IN1702_I
          input  IN1703_I : IN_DIGITAL_A_INPUT_MAPPING_TYPE  // IN1703_I
          input  IN1800_I : IN_DIGITAL_A_INPUT_MAPPING_TYPE  // IN1800_I
          input  IN1801_I : IN_DIGITAL_A_INPUT_MAPPING_TYPE  // IN1801_I
          input  IN1802_I : IN_DIGITAL_A_INPUT_MAPPING_TYPE  // IN1802_I
          input  IN1803_I : IN_DIGITAL_A_INPUT_MAPPING_TYPE  // IN1803_I
          input  IN0300_I : IN_DIGITAL_B_INPUT_MAPPING_TYPE  // IN0300_I
          input  IN0301_I : IN_DIGITAL_B_INPUT_MAPPING_TYPE  // IN0301_I
          input  IN0800_I : IN_DIGITAL_B_INPUT_MAPPING_TYPE  // IN0800_I
          input  IN0801_I : IN_DIGITAL_B_INPUT_MAPPING_TYPE  // IN0801_I
          input  IN1300_I : IN_DIGITAL_B_INPUT_MAPPING_TYPE  // IN1300_I
          input  IN1301_I : IN_DIGITAL_B_INPUT_MAPPING_TYPE  // IN1301_I
          input  IN1302_I : IN_DIGITAL_B_INPUT_MAPPING_TYPE  // IN1302_I
          input  IN1303_I : IN_DIGITAL_B_INPUT_MAPPING_TYPE  // IN1303_I
          input  COM_RESET_I : IN_COMMUNICATION_RESET_INPUT_MAPPING_TYPE  // COM_RESET_I
          input  IN0000_I : IN_FREQUENCY_B_CHANNEL_A_INPUT_MAPPING_TYPE  // IN0000_I
          input  IN0002_I : IN_FREQUENCY_B_CHANNEL_A_INPUT_MAPPING_TYPE  // IN0002_I
          input  IN0500_I : IN_FREQUENCY_B_CHANNEL_A_INPUT_MAPPING_TYPE  // IN0500_I
          input  IN0502_I : IN_FREQUENCY_B_CHANNEL_A_INPUT_MAPPING_TYPE  // IN0502_I
          input  IN1000_I : IN_FREQUENCY_B_CHANNEL_A_INPUT_MAPPING_TYPE  // IN1000_I
          input  IN1002_I : IN_FREQUENCY_B_CHANNEL_A_INPUT_MAPPING_TYPE  // IN1002_I
          input  IN1500_I : IN_FREQUENCY_B_CHANNEL_A_INPUT_MAPPING_TYPE  // IN1500_I
          input  IN1502_I : IN_FREQUENCY_B_CHANNEL_A_INPUT_MAPPING_TYPE  // IN1502_I
          input  IN0001_I : IN_FREQUENCY_B_CHANNEL_B_INPUT_MAPPING_TYPE  // IN0001_I
          input  IN0003_I : IN_FREQUENCY_B_CHANNEL_B_INPUT_MAPPING_TYPE  // IN0003_I
          input  IN0501_I : IN_FREQUENCY_B_CHANNEL_B_INPUT_MAPPING_TYPE  // IN0501_I
          input  IN0503_I : IN_FREQUENCY_B_CHANNEL_B_INPUT_MAPPING_TYPE  // IN0503_I
          input  IN1001_I : IN_FREQUENCY_B_CHANNEL_B_INPUT_MAPPING_TYPE  // IN1001_I
          input  IN1003_I : IN_FREQUENCY_B_CHANNEL_B_INPUT_MAPPING_TYPE  // IN1003_I
          input  IN1501_I : IN_FREQUENCY_B_CHANNEL_B_INPUT_MAPPING_TYPE  // IN1501_I
          input  IN1503_I : IN_FREQUENCY_B_CHANNEL_B_INPUT_MAPPING_TYPE  // IN1503_I
    Communication : Communication, ifm electronic, version 3.1.4.1
      Ethernet : Ethernet, ifm electronic, version 3.1.4.1
      CAN : CAN, ifm electronic, version 3.1.4.1
  CR721S : CR721S, ifm electronic, order no. CR721S, version 3.1.4.1
  Project Information/
    function GetVersion [ST]
    function GetCompany [ST]
    function GetTitle [ST]
    function GetTextProperty2 [ST]
    function GetTextProperty [ST]
    function GetBooleanProperty [ST]
    function GetVersionProperty [ST]
    function GetNumberProperty [ST]
*)

// StandardPLC/Application/FIFO_DUT
TYPE FIFO_DUT :
STRUCT
	New:UINT;
	CurrentNum:UINT;
	FirstElement:UINT;
	Element:ARRAY[0..30] OF UINT;
	WR:BOOL;
	WR_1:BOOL;
	RD:BOOL;
	RD_1:BOOL;
END_STRUCT
END_TYPE

// StandardPLC/Application/GLV/PersistentVars
VAR_GLOBAL PERSISTENT RETAIN
	(*深度参数*)
	Par_Save_Depth :INT:=0;
	Tmp_Depth :INT;
	PAR_DEPTH_accumu: UDINT:=0;
	Mid_Depth_Accumu :UDINT;
	Depth_Accumu :UDINT;
	DEPTH:INT;
	PAR_DEPTH_VALUE:UINT;
	PAR_DEPTH_VALUE2:UINT;
	(*燃油消耗量*)
	tmp_FUEL: UDINT;
	Par_Accumu_Fuel_1: UDINT:=0;
	
(*GPS*)
	VarCanNewGpsVersion:UINT;//通讯协议版本号
	VarCanNewGpsManufacturers:USINT;//GPS厂家类别
	VarGpsTempUnlockPassword:UINT;//临时解锁密码
	VarGpsYongJiuUnlockPassword:DINT;//永久解锁密码
	VarGpsYongJiuUnlockPassword2:DINT;//永久解锁密码2
	VarGpsGlobalEnable:BOOL:=TRUE;//GPS全局使能    1-GPS锁车有效 0-已永久解锁
	VarGpsTempUnlockDoing:BOOL:=FALSE;//临时解锁使能   0-GPS锁车有效 1-已临时解锁
	VarGpsSystemLockedState:BOOL;//系统锁机标志 0-未锁车  1-锁车 
	VarCanNewGpsRecLockCommand:USINT;
	VarCanNewGpsRecUnlockCommand:USINT;
	VarGpsPasswordTempUnlockEnable:BOOL; //GPS密码临时解锁使能
	VarGpsPasswordTempUnlockCount:USINT;//控制器连续收到GPS验证临时解锁密码结果正确的次数
	VarGpsPasswordTemporaryCode:UDINT;//GPS临时解锁密码值（11个每个只能使用一次）
	VarCanNewGpsRealFakeRecData:UINT;//真假GPS识别数据
	VarCanNewGpsRealFakeTargetData:UINT;//真假GPS识别目标数据
	VarCanNewGpsRealFakeResult:BOOL;//真假GPS识别
	CAN_NewGpsRealFakeTranData:UINT;//随机发送的数据
	VarGpsPasswordTempUnlockTimer60S:UINT;//临时解锁计时
	VarGpsPasswordUlockCancle:BOOL;//
	VarCanGpsTongXunLockErrorTimer2S:UINT;//GPS总线故障计时
	VarCanGpsFakeErrorTimer1S:UINT;//假GPS计时
	VarGpsTempUnlockSelect:USINT;//GPS临时解锁选择位
	VarGpsTempUnlockEnable:USINT:=16#FF;//GPS临时解锁使能位
	GPS_Time_Year_Last: USINT;
	GPS_Time_Month_Last: USINT;
	GPS_Time_Day_Last: USINT;
	GPS_Time_Hour_Last: USINT;
	GPS_Time_Minute_Last: USINT;
	GPS_Time_Second_Last: USINT;
	Time_bool_once:BOOL:=TRUE;
	Time_bool_once2:BOOL:=TRUE;
	GPS_Time_Year_Last2: USINT;
	GPS_Time_Month_Last2: USINT;
	GPS_Time_Day_Last2: USINT;
	GPS_Time_Hour_Last2: USINT;
	GPS_Time_Minute_Last2: USINT;
	GPS_Time_Second_Last2: USINT;
	VarGpsSystemLockedState_bool :BOOL;	
	PAR_GPS_TempUnlockPassword:UDINT;
	PAR_GPS_ForeverUnlockPassword:DINT;
	VarCanGpsKongZhiQiLockCommand:BOOL;//来自Gps的锁车指令
	VarCanGpsYanShiLockCommand:BOOL;//GPS故障锁车1=7天无信号
	VarCanGpsTianXianLockCommand:BOOL;//GPS故障锁车2=天线故障
	VarCanGpsKaiGaiLockCommand:BOOL;//GPS故障锁车3=盒盖打开
	VarCanGpsTongXunLockCommand:BOOL;//GPS故障锁车4=拆除GPS
	VarCanGpsFakeLockCommand:BOOL;//GPS故障锁车5=假GPS
	VarcanGPSbakaCommand:BOOL;//GPS故障锁车6=拔卡故障
	VarCanGpsYanShiLockCommand_Enable:BOOL:=TRUE;(*GPS故障锁车1=7天无信号*)(*盲区*)
	VarCanGpsBakaLockCommand_Enable:BOOL:=TRUE;(*GPS故障锁车2=天线故障*)(*拔卡*)
	VarCanGpsKaiGaiLockCommand_Enable:BOOL:=TRUE;(*GPS故障锁车3=盒盖打开*)(*拆盖*)
	VarCanGpsTongXunLockCommand_Enable:BOOL:=TRUE;(*GPS故障锁车4=拆除GPS*)(*总线*)
	VarCanGpsenableALLLockCommand:BOOL:=TRUE;(*来自Gps的总使能锁车指令*)
	VarCanGpsBEIDONGLockCommand:BOOL:=TRUE;(*来自Gps的被动锁车指令*)
	VarCanGpsYanShiLockCommand_time:UINT:=480;(*20天无信号锁车*)(*480/24=20*)
	Varjilu_PAR_WorkTime:UDINT;(*记录的工作时间*)
	Varjilu_PAR_WorkTime2:UINT;(*延时6小时锁车时间*)
		
	
(*工作时间参数*)
	Mid_worktime			: UDINT;
	PAR_worktime            : UDINT;
(*备用*)
	PAR_GLB_max:UINT:=50;(*高怠速时泵的吸收功率*)
	PAR_GLB_min:UINT:=5;(*低怠速时泵吸收功率*)
	PAR_GLB_66:UINT:=48;(*转速为66%时泵的吸收功率*)
	PAR_GLB_33:UINT:=40;(*转速为33%时泵的吸收功率*)
(*桅杆参数*)
	PAR_Zero_AngleX:UINT:=32767;
	PAR_Zero_AngleY:UINT:=32767;
(*PID参数*)
	PAR_PID_ENABLE								:BOOL:=TRUE;
	PAR_CYCLE								:UINT:=2;(*hmi*)
	PAR_RC									:USINT:=10;(*hmi*)
	PAR_OUT_UP									:INT:=32767;
	PAR_OUT_DWN									:INT:=-32767;
	PAR_SV									:UINT:=100;
	lever_ok													: BOOL;
	
(***************显示屏设置参数******************)

(*步长参数*)
	PAR_ControlValue:UINT:=10000;
(*主参数*)
	PAR_Circle1 :UINT:=980;(*hmi毫米*)(*外圈直径*)
	PAR_Circle2 :UINT:=980;(*hmi毫米*)(*内圈直径*)
	Par_Circle3: UINT;
	PAR_Quanshu : UINT:=25;(*hmi圈*)
(*参数设置*)
	PAR_MainAngleSetting:UINT:=10;
	PAR_RotationPercision:UINT;
	PAR_Speed_Idling:UINT:=1000;
(*泵参数*)
	PAR_SpeedLow_Idling:UINT:=1000;
	PAR_SpeedHigh_Idling:UINT:=1900;
	PAR_Pump1Current_Max:UINT:=1000;
	PAR_Pump1Current_Min:UINT:=0;
	PAR_Pump2Current_Max:UINT:=1000;
	PAR_Pump2Current_Min:UINT:=0;
(*手柄设置界面*)
	Par_Joy_DeadBand:UINT:=60;(*手柄死区*)
	Par_Joy_DeadBand_max: UINT:=20;(*手柄阶跃死区*)
	PAR_NegFull_x : UINT:=380;  //1450 恒功率点
	PAR_PosFull_x : UINT:=380; //1600 恒功率点
	PAR_Zero_x    :UINT:=350;  //1800 恒功率点
	PAR_DeadBand_x :UINT:=10; //功率控制时间	
	PAR_Progression_x  :UINT;
	PAR_NegFull_y : UINT:=150;//1450  加载时间
	PAR_PosFull_y : UINT:=150;//1600  加载时间
	PAR_Zero_y    : UINT:=200; //1800  加载时间
	PAR_DeadBand_y  : UINT;
	PAR_Progression_y  : UINT;
	PAR_M_Joy_LEN:UINT;
(*回转设置界面*)
	PAR_Sudu1_Min:UINT:=3000;
	PAR_Sudu1_Max:UINT:=5000;
	PAR_Sudu1_Middle:UINT:=4000;
	PAR_Angle1:UINT:=4;
	PAR_Angle2:UINT:=510;
	PAR_Angle3:UINT:=100;
	PAR_Angle4:UINT:=4094;
	PAR_Angle5:UINT:=3580;
	PAR_Angle6:UINT:=3990;
	PAR_Sudu2_Min:UINT:=3000;
	PAR_Sudu2_Max:UINT:=5000;
	PAR_Sudu2_Middle:UINT:=4000;
(*报警设置界面*)
	PAR_WarnFuelLevel_Low:UINT:=15;
	PAR_WarnHydOilTem_High:UINT:=90;
	PAR_WarnOilPress_Low:UINT:=20;
	PAR_WarnWaterTem_High:UINT:=100;
	PAR_HydOilPress_PosFull:UINT:=20000;
	PAR_HydOilPress_NegFull:UINT:=4000;
	PAR_HydOilPilotPress_PosFull:UINT:=20000;
	PAR_HydOilPilotPress_NegFull:UINT:=4000;
	PAR_TensionSensor_PosFull:UINT:=20000;
	PAR_TensionSensor_NegFull:UINT:=4000;
	PAR_TensionSensor_Range:UINT:=40;
	PAR_WarnTension_High:UINT:=200;	
	Par_Tension_coe: REAL:=0.6;

(*PID电比例阀设置*)
	PAR_KP:UINT:=550;  //副卷速度调节
	PAR_KI:BYTE:=45; //复合动作动力头速度调节
	PAR_KD:BYTE:=2;//1:p+g手柄   2：恒力手柄
	PAR_Y27_PosFull:UINT:=630;(*阀A正向*)
	PAR_Y27_NegFull:UINT:=300;
	PAR_Y28_PosFull:UINT:=550;(*阀A逆向*)
	PAR_Y28_NegFull:UINT:=300;
	PAR_Y29_PosFull:UINT:=630;(*阀B正向*)
	PAR_Y29_NegFull:UINT:=300;
	PAR_Y30_PosFull:UINT:=550;(*阀B逆向*)
	PAR_Y30_NegFull:UINT:=300;	
(*阀D加压限压参数*)
	PAR_ValveD_PosFull:UINT:=510;  //加压限制
	PAR_ValveD_NegFull:UINT:=300;  //冷却风扇
(*阀C加压限压参数*)
	PAR_ValveC_PosFull:UINT:=500;  //抛土
	PAR_ValveC_NegFull:UINT:=650;	//回转
(*主泵*)
	PAR_Valve1_PosFull:UINT:=1300;
	PAR_Valve1_NegFull:UINT:=500;
	PAR_Valve2_PosFull:UINT:=1300;
	PAR_Valve2_NegFull:UINT:=500;
	PAR_Valve3_PosFull:UINT:=800;
	PAR_Valve3_NegFull:UINT:=300;
	PAR_Valve4_PosFull:UINT:=1300;
	PAR_Valve4_NegFull:UINT:=1000;
	PAR_Valve5_NegFull:UINT:=600;
	PAR_Y1_PosFull:UINT:=700;
	PAR_Y1_NegFull:UINT:=400;
	PAR_Y1_1_PosFull:UINT:=700;
	PAR_Y1_1_NegFull:UINT:=300;
	PAR_Y2_PosFull:UINT:=700;
	PAR_Y2_NegFull:UINT:=400;
	PAR_Y3_PosFull:UINT:=700;  
	PAR_Y3_NegFull:UINT:=300; 
	PAR_Y4_PosFull:UINT:=500;
	PAR_Y4_NegFull:UINT:=200;
	PAR_Y5_PosFull:UINT:=500;
	PAR_Y5_NegFull:UINT:=200;
	PAR_Y6_PosFull:UINT:=500;
	PAR_Y6_NegFull:UINT:=200;
(*液压功能选择界面*)
	PAR_MainPumpChioce:BYTE:=1;
	PAR_M4ValveChioce:BYTE:=1;
	PAR_MotorChioce:BYTE:=1;

(*主卷带杆报警界面*)
	PAR_ChuDi_High: UINT;
	PAR_MainWinchLaLi_Low:UINT:=2000;
	PAR_DrillWeight1:UINT;
	PAR_DrillWeight2:UINT;
	PAR_DrillWeight3:UINT;
	PAR_DrillWeight4:UINT;
	PAR_DrillWeight5:UINT;
	PAR_DrillWeightOriginal:UINT;
(*加压卷扬设置界面*)
	PAR_JiYaWinch_Diameter:UINT:=355;
(*左右限位标定值*)
	PAR_L_LimiteValue:UINT:=1900;
	PAR_R_LimiteValue:UINT:=3100;
(*油门标定界面*)
	PAR_YouMen_NegFull:UINT:=920;
	PAR_YouMen_PosFull:UINT:=3400;	
(*加压台显示设置*)
	PAR_ZhuangGan_Number:UINT:=0;
	PAR_BianFu_Location:UINT:=2000;
	PAR_ZuanTong_Location:UINT:=1500;	
(*动力头变量*)
	PAR_MotorChioce_H_PWM:UINT:=590;
	PAR_MotorChioce_M_PWM:UINT:=380;
	PAR_MotorChioce_L_PWM:UINT:=10;
	
	(*节能状态（打开或关闭)*)
	SaveEngineState:BOOL;
END_VAR

// StandardPLC/Application/SaveEngine/GVL_SaveEngine

VAR_GLOBAL
	(*节能*)
	AcDecompression:BOOL:=FALSE;//泄压模式
	SaveEngineMode:UINT:=0;//节能模式
	
	//AI_PAcPreMv:UINT;(* B36 IN1600 节能蓄能器油压,单位毫伏*)
	//AI_PAtomsPreMv:UINT;(* B37 IN1601 节能蓄能器气压,单位毫伏*)
	AI_PAcPreMv:UINT;(* B36 IN1600 节能蓄能器油压,单位毫伏*)
	AI_PAtomsPreMv:UINT;(* B37 IN1601 节能蓄能器气压,单位毫伏*)
	
	AI_PM1PreMv:UINT;(*B38节能M1压力下放马达出口,单位毫伏*)
	AI_PM2PreMv:UINT;(*B39节能M2压力下放马达入口,单位毫伏*)
	
    AI_PAcPre:UINT;(* IN1600 节能蓄能器油压*)
	AI_PAtomsPre:UINT;(* IN1601 节能蓄能器气压*)
	AI_PM1Pre:UINT;(*节能M1压力下放马达出口,BAR*)
	AI_PM2Pre:UINT;(*节能M2压力下放马达入口,BAR*)
	
	Y72OutPutState:BOOL:=FALSE;(*B66*)
	Y71OutPutState:BOOL:=FALSE;(*B76*)
	Y73:BOOL:=FALSE;(*B78*)
	Y74:BOOL:=FALSE;(*B71*)
	//DT3OutPutState:BOOL:=FALSE;

	Rotation_move: BOOL;
	MainWinch_move:BOOL;
	PowerHead_move:BOOL;
	JiaYa_move: BOOL;
	ViceWinch_move: BOOL;
	LeftMove_move:BOOL;
	RightMove_move:BOOL;
	DOH_Y50_1: BOOL;//0
	
	SPEED_CASE:USINT;//GLV
	Enginer_Power:UINT;//GLV
	PWM_Y1_Target: UINT:=0;	//GLV
	PWM_Y2_Target: UINT:=0;	//GLV
	MainPump_Pressure_Taget:UINT;	//GLV
	MainPump_Pressure: UINT;//GLV
	Pressure_Coe: REAL;//GLV
	PWM_Y1_Target_OutPut: UINT;//GLV
	PWM_Y2_Target_OutPut: UINT;//GLV
	PWM_Y33_SET_Target: UINT:=1100;//GLV
	MainPump_Pressure_Taget1000:UINT:=180;//GLV
	MainPump_Pressure_Taget1200:UINT:=260;//GLV
	MainPump_Pressure_Taget1450:UINT:=450;//GLV
	MainPump_Pressure_Taget1600:UINT:=430;//GLV
	MainPump_Pressure_Taget1750:UINT:=430;//GLV
	MainPump_Pressure_Taget1900:UINT:=400;//GLV	
	Pressure_Coe_Taget: REAL;//GLV
	JianGE1: REAL:=1;//GLV
	JianGE2: REAL:=0.005;//GLV
	TIME_100ms:TON;//GLV

	MainPump_Pressure_last1: UINT;//GLV
	TIME_LvBo1:TON;//GLV
	TIME_LvBo2:TON;//GLV
	MainPump_Pressure_Subtract: INT;//GLV
	MainPump_Pressure_ChangeBool: BOOL;//GLV
	MainPump_Pressure_ChangeBool1:BOOL;//GLV
	EngineSpeedSub: UINT;//GLV
	ECO_Press_Target1000: UINT:=50;
	ECO_Press_Target1200: UINT:=50;
	ECO_Press_Target1400: UINT:=50;
	ECO_Press_Target1600: UINT:=50;
	ECO_Press_Target1800: UINT:=50;
	ECO_Press_Target1900: UINT:=50;
	
	HELIU_Press_Target1000: UINT:=50;
	HELIU_Press_Target1200: UINT:=50;
	HELIU_Press_Target1400: UINT:=100;
	HELIU_Press_Target1600: UINT:=100;
	HELIU_Press_Target1800: UINT:=100;
	HELIU_Press_Target1900: UINT:=100;
	BiaoZHI_MainWinchUp: BOOL;//GLV
	JianGE6:REAL:=2;//GLV
	PWM_Y8_SET_Target: UINT;//GLV
	PWM_Y10_SET_Target: UINT;//GLV
	PWM_Y7_SET_Target: UINT;//GLV
	PWM_Y9_SET_Target: UINT;//GLV
	PWM_Y8_SET_Target1: INT;//GLV
	PWM_Y10_SET_Target1: INT;//GLV
	PWM_Y7_SET_Target1: INT;//GLV
	PWM_Y9_SET_Target1: INT;//GLV
	Joyx_change_bool: BOOL;//GLV
	curve7:curve_quxian;//GLV
	curve8:curve_quxian;//GLV
	curve9:curve_quxian;//GLV
	curve10:curve_quxian;//GLV
	curve19:curve_quxian;
	curve20:curve_quxian;

	TIMEBASE:TIME:=T#200MS;//GLV
	RAMP7:RAMP_INT;//GLV
	RAMP8:RAMP_INT;//GLV
	RAMP9:RAMP_INT;//GLV
	RAMP10:RAMP_INT;//GLV
	RAMP15:RAMP_INT;//GLV
	RAMP16:RAMP_INT;//GLV
	RAMP19:RAMP_INT;
	RAMP20:RAMP_INT;
	RAMP21:RAMP_INT;

	//2023 01 13 增加
	//动力头动作斜坡值
	R_RAMP_ratate:INT:=800;
	F_RAMP_ratate:INT:=400;
	TIMEBASE_ratate:TIME:=T#100MS;
	//主卷扬动作斜坡值
	R_RAMP_mainwinch:INT:=800;
	F_RAMP_mainwinch_up:INT:=400;
	F_RAMP_mainwinch_down:INT:=400;
	TIMEBASE_mainwinch:TIME:=T#200MS;
	//主泵排量斜坡值
	R_RAMP_pump:INT:=300;
	F_RAMP_pump:INT:=1000;
	TIMEBASE_pump:TIME:=T#1000MS;
	Subtract: BOOL;//GLV
	TIME_LvBo4:TON;//GLV
	Curve_input:UINT;//GLV
	Curve_Par: SINT:=0;//GLV
	PWM_Y39_SET1:UINT;//GLV
	PWM_Y40_SET1:UINT;//GLV
	PWM_Y9_SET1:INT;//GLV
	PWM_Y10_SET1:INT;//GLV
	PWM_Y13_SET1:INT;//GLV
	PWM_Y14_SET1:INT;//GLV
	yanchi1:BOOL;//GLV
	yanchi_ton1:ton;//GLV
	RAMP15_IN:UINT;//GLV
	RAMP16_IN:UINT;//GLV
	PWM_Y39_SET_Target: UINT;
	PWM_Y40_SET_Target: UINT;
	Curve_Par1: SINT:=0;	
	PWM_Y39_SET_Target1:INT;
	PWM_Y40_SET_Target1:INT;
	PWM_Y37_SET_Target:UINT;
	PWM_Y17_SET2:UINT;
	t_PowerHead_move:TON;
	x_t_PowerHead_move:INT:=10;//100-10
	x2_t_PowerHead_move:INT:=10;//100-10

		//卸荷阀斜坡值
	R_RAMP_xiehe:INT:=800;
	F_RAMP_xiehe:INT:=400;
	TIMEBASE_xiehe:TIME:=T#500MS;
	
	//直线阀斜坡值
	R_RAMP_zhixian:INT:=800;
	F_RAMP_zhixian:INT:=800;
	TIMEBASE_zhixian:TIME:=T#300MS;

	OLength :UINT :=1200;//GLV 一节钻杆长度,cm
	
//	TIME_1000ms_ESDownStart:TON;//GLV
	PWM_JOYY_L_UP_1: INT;// GLV  手柄信号中间变量 
	JoyDesFlag:BOOL:=FALSE;//松手柄标志
	JoyDesTimer:UINT;
	JoyDesto0_flag :BOOL :=FALSE;//GLV
	Mode2Timer:UINT;
	Mode1Timer:UINT;
	Mode1Timer_1:UINT;
	Mode4Timer: UINT;
	Mode7Timer:UINT;
	Mode8Timer: UINT;
	Mode10Timer: UINT;
	Mode12Timer: UINT;
	Mode11Timer: UINT;
	Rtrig_DongLiTou1:R_TRIG;
	Rtrig_DongLiTou2:R_TRIG;
	Count_TIMES_Fanzhuan: UINT;
	Count_TIMES_Zhengzhuan: UINT;
	TIME_1000ms:TON;
	TIME_1000ms_TP:TON;
	Count_TIMES_Fanzhuan_LAST: UINT;
	Count_TIMES_Zhengzhuan_LAST: UINT;
	Paotu_Modle: BOOL;
	PaoTU_biaozhi: BOOL;
	TIMEBASE_D: TIME;
	
	P25_Flag:BOOL;
	P27_Flag:BOOL;
	P29_Flag:BOOL;
	P31_Flag:BOOL;
	
	MainWinchTension_Ave: REAL;
	t_powertime:TIME;
	Max_MainWinchTension:REAL;
//	PWM_Y33_SET_Target: UINT:=370;//主卷目标电流	

END_VAR

// StandardPLC/Application/GLV/Global_Variablen

VAR_GLOBAL
	init_1				: BOOL :=TRUE;
	init_2				: BOOL :=TRUE;
	
(*倾角*)
	delta_x				: INT;
	delta_y				: INT;
(*限位*)
	TooLowX_angle		: BOOL;
	TooHighX_angle		: BOOL;
	TooHighY			: BOOL;
(*回转*)
	CANO_ZHIXING     	:BOOL;
	PI_Rotation_COUNTER	:DINT;
	PI_ROTATE_VALUE		:UINT;
	AUTO_ROTATION_VALVE: INT;
(*深度计算*)
	PI_Depth_COUNTER	:DINT;
	VarDepthLastMax: UINT:=1000;
	VarMaiWinDepth_subtract:DINT;
	VarMaiWinDepth_Up_biaozhi: BOOL;
	VarMaiWinDepthLast: UINT:=1000;
	VarMaiWinDepthOnce: UINT;
	VarMaiWinDepthTotal: UINT;
	
	IncEncoder_temp_diValue:DINT;
	CW: BOOL;
	CCW: BOOL;
	temp_f:REAL;
	A_DEEP:BOOL;
	
	

(*提升限位取消*)
	PAR_DISTANCE_CANCEL								:BOOL;(*hmi*)
	
(*桅杆控制*)	
	VarMastA_			:INT;
	VarMastB_			:INT;
	VarMastA			:INT;
	VarMastB			:INT;
	VarJoyY 			:INT;
	VarJoyX				:INT;
	VarJoyY100			:INT;
	VarJoyX100			:INT;
	VarGama				:UINT:=90;
	VarLengthC			:REAL;
	VarAngleXDelta		:INT;
	VarAngleYDelta		:INT;	
	VarMastAutoEnable	:BOOL;
	VarMastManuEnable	:BOOL;
	CANI_Button_LEVER_AutoLast	:BOOL;
	CANI_Button_LEVER_ManualLast:BOOL;
	VarMastLimitCancel	:BOOL;
	VarMastLimitState	:UINT;
	VarMastWorkMode :UINT;
(*平均值*)
	mean1:FIFO_DUT;
    mean2:FIFO_DUT;
    mean3:FIFO_DUT;
    mean4:FIFO_DUT;	
    mean5:FIFO_DUT;	
(*发动机转速*)
	EngineSpeedTarget:UINT;
(*燃油消耗*)
	CANO_Accumu_Fuel_2: UDINT;	
	FuelMomentary: UINT;
	FuelMomentary1: UINT;
(*施工参数*)
	PileDiameter: UINT;
	PileNumble: UDINT;
	CANO_PowerSpeed: UINT;
	CANO_PowerNiuJu: UINT;	
	CANO_X_PIANYIZHI:UINT;
	CANO_Y_PIANYIZHI:UINT;
	
	reset111: BOOL;	
	UIGroupVoltage0: UINT;
	UIGroupVoltage1: UINT;
	UIGroupVoltage2: UINT;
	UIGroupVoltage3: UINT;
	UIGroupVoltage4: UINT;
	UIGroupVoltage5: UINT;
	
	
	(*GPS统型协议*)
	
	VarCanGpsLockCommand_A:BOOL;(*来自Gps的A锁车指令*)
	VarCanGpsLockCommand_B:BOOL;(*来自Gps的B锁车指令*)
	VarCanGpsLockCommand_C:BOOL;(*来自Gps的C锁车指令*)
	VarCanGpsLockCommand_D:BOOL;(*来自Gps的D锁车指令*)
	VarCanGpsLockCommand_E:BOOL;(*来自Gps的E锁车指令*)
	VarCanGpsJIAOYANNUM:UINT;(*接收Gps真伪校验序列号*)
	VarCanGpsJIAOYANMA:UINT;(*接收Gps真伪校验码*)

	VarCANGPSYINGDAREC_ID:UINT;(*Gps应答接收ID*)
	VarCANGPSYINGDAREC_DATA:UINT;(*Gps应答接收数据*)
	VarCANGPSYINGDASEND_ID:UINT;(*Gps应答发送ID*)
	VarCANGPSYINGDASEND_DATA:UINT;(*Gps应答发送数据*)

	Senddata_2FF:ARRAY [0..5] OF BYTE;(*真伪校验参数*)
	Ver_Result:UINT;

	data_2FF:ARRAY [0..5] OF BYTE;(*真伪校验参数*)
	uLength01:BYTE;
	Ver_Output:UINT;
	GPS_Lock_Beidong:BOOL;	
	
		(*GPS延时锁车*)
	VarCanNewGpsNoSignalLock_Warning: BOOL;	
	VarCanNewGpsNoSignalLock_Warning2:BOOL;
	STATE_Promoteconnect_20day_2:BOOL;
	GPS_Time_bool: BOOL;
	GPS_Time_Year: USINT;
	GPS_Time_Month: USINT;
	GPS_Time_Day: USINT;
	GPS_Time_Hour: USINT;
	GPS_Time_Minute: USINT;
	GPS_Time_Second: USINT;
	GPS_Signal_Intensity: USINT;
	Time_Minute_Left: UINT;
	Time_Sub_Year: USINT;
	Time_Sub_Month: USINT;
	Time_Sub_Day: USINT;
	Time_Sub_Hour: USINT;
	Time_Sub_Minute: USINT;
	Time_Sub_Second: USINT;
	Time_Sub_Year2: SINT;
	Time_Sub_Month2: SINT;
	Time_Sub_Day2: SINT;
	Time_Sub_Hour2: SINT;
	Time_Sub_Minute2: SINT;
	Time_Sub_Second2: SINT;
	Time_Minute_Left2: DINT;
	Time_hour_Left2:DINT;
	
	VarGpsTempUnlockPassword2:DINT;//临时解锁密码2
	
	CANO_DONGTAIMA1:DINT;
	CANO_DONGTAIMA2:DINT;
	
	
	//国四发动机
	ZAISHENG_LIGHT:BOOL;
	JINZHI_LIGHT:BOOL;
	GAOPAIWEN_LIGHT:BOOL;
	DEF_LIGHT:BOOL;
	JIASHIYUANWARN_LIGHT:BOOL;
	urea_level:BYTE;
	VarZaishengjinzhiSwitch:BOOL;
	VarHouchuliSwitch:BYTE;
	VarQiangzhiZaishengSwitch:BOOL;
	
	M2_Press_H_C:BOOL;
END_VAR

// StandardPLC/Application/GLV/IO_GLV
VAR_GLOBAL
	(*IO端口*)
	
	(*A端口*)
	(***********输入************)
	(*PI*)
	PI_SP2A:UDINT;(*A25 回转编码器A*)
	PI_SP2B:UDINT;(*A26 回转编码器B*)
	PI_SQ1:UDINT;(*A27 深度*)
	PI_SQ2:UDINT;(*A28 深度*)
	(*DIH*)
	DIH_SQ1:BOOL;  (*A27 深度接近开关SQ1*)
	DIH_SQ2:BOOL;  (*A28 深度接近开关SQ2*)
	DIH_JOY:BOOL;  (*A36 立桅杆电手柄JOY*)
	DIH_SA8:BOOL;  (*A37 浮动脚踏开关SA8*)
	DIH_SP4:BOOL;  (*A38 回油滤芯开关SP4*)
	DIH_SQ12:BOOL; (*A39 平举限位开关SQ12*)
	DIH_SQ5:BOOL;  (*A44 桅杆左限位开关SQ5*)
	DIH_SQ6:BOOL;  (*A45 桅杆右限位开关SQ6*)
	DIH_SQ8:BOOL:=TRUE;  (*A46 重锤上限位SQ8*)
	DIH_SA18:BOOL;(*A47  动力头慢速*)
	DIH_SA19:BOOL;(*A70  行走快速*)
	DIH_SA15:BOOL;(*B6  动力头限扭*)
	DIH_power3:BOOL;(*B10  钥匙开关*)
	
	(*DIL*)
	DIL_SQ3:BOOL;  (*A40 先导开关SQ3*)
	DIL_SQ4:BOOL;  (*A41 主卷上限位开关SQ4*)
	DIL_SQ11:BOOL; (*A42 动力头上限位开关SQ11*)
	DIL_SQ13:BOOL; (*A43 液压油位开关SQ13*)
	
	(*AI*)
	AI_P1:UINT;    (*A55 加压压力P1*)
	AI_P2:UINT;    (*A56 动力头压力P2*)
	AI_P3:UINT;    (*A57 主卷压力P3*)
	AI_P11:UINT;   (*A58 主泵1压力P11*)
	AI_P12:UINT;   (*A59 主泵2压力P12*)
	AI_P6:UINT;    (*A60 副泵压力P6*)
	AI_P7:UINT;    (*A61 先导压力P7*)
	AI_JOYX:UINT;  (*A62 立桅杆电手柄JOYX*)
	AI_JOYY:UINT;  (*A63 立桅杆电手柄JOYY*)
	AI_SP1:UINT;   (*A64 燃油液位SP1*)
	AI_SP1_1: UINT;
	AI_SP3:UINT;   (*A65 液压油温SP3*)
	AI_SP3_1:UINT;(*限制*)
	AI_SP7:UINT;   (*A66 销轴传感器SP7*)
	AI_SP11:UINT;  (*A67 左右倾角角度传感器*)
	AI_ECM2_9:UINT;(*A68 油门旋钮ECM2_9*)
//	AI_AngleX:UINT;(*A69 倾角传感器X向 AngleX*)
//	AI_AngleY:UINT;(*A70 倾角传感器Y向 AngleY*)
	AI_P1A:UINT;   (*A69 加压压力P1A*)
	
	
    (***********输出************)
	(*PWM*)
	PWM_Y1:UINT;   (*A06 主泵1调节Y1*)
	PWM_Y1_SET:INT;
	PWM_Y3:UINT;   (*A07 副卷上Y3*)
	PWM_Y3_SET:UINT;
	PWM_Y2:UINT;   (*A16 主泵2调节Y2*)
	PWM_Y2_SET:INT;
	PWM_Y4:UINT;   (*A09 副卷下Y4*)
	PWM_Y4_SET:UINT;
	PWM_Y5:UINT;   (*A10 左行走前进Y5*)
	PWM_Y5_SET:UINT;
	PWM_Y17:UINT;  (*A11 加压快上提Y17*)
	PWM_Y17_SET:UINT;(*A11 加压快上提Y17*)
	PWM_Y33:UINT;  (*A12 主卷变量控制Y33*)
	PWM_Y33_SET:UINT;
	PWM_Y45:UINT;  (*A13 绳张紧缩*)
	PWM_Y45_SET:UINT;
	PWM_Y18:UINT;  (*A14 加压快下放Y18*)
	PWM_Y18_SET:UINT;(*A14 加压快下放Y18*)
	PWM_Y6:UINT;   (*A08 左行走后退Y6*)
	PWM_Y6_SET:UINT;	
	PWM_Y19:UINT;  (*A17 履带伸Y19*)
	PWM_Y19_SET:UINT;
	PWM_Y9:UINT;   (*A18 主卷2上提Y9*)
	PWM_Y9_SET:UINT;
	PWM_Y20:UINT;  (*A19 履带缩Y20*)
	PWM_Y20_SET:UINT;
	PWM_Y10:UINT;  (*A20 主卷2下放Y10*)
	PWM_Y10_SET:UINT;
	PWM_Y23:UINT;  (*A21 加压下Y23*)
	PWM_Y23_SET:UINT;
	PWM_Y7:UINT;   (*A22 主卷上提Y7*)
	PWM_Y7_SET:UINT;
	PWM_Y8:UINT;   (*A23 主卷下放Y8*)
	PWM_Y8_SET:UINT;	
	PWM_Y11:UINT;  (*A24 动力头2正转Y11*)
	PWM_Y11_SET:UINT;
	PWM_Y12:UINT;  (*A73 动力头2反转Y12*)
	PWM_Y12_SET:UINT;	
	PWM_Y24:UINT;  (*A74 加压上Y24*)
	PWM_Y24_SET:UINT;
	PWM_Y15:UINT;  (*A75 右行走前进Y15*)
	PWM_Y15_SET:UINT;
	PWM_Y25:UINT;  (*A76 变幅伸出Y25*) 
	PWM_Y25_SET:UINT;
	PWM_Y16:UINT;  (*A77 右行走后退Y16*)
	PWM_Y16_SET:UINT;
	PWM_Y26:UINT;  (*A78 变幅缩回Y26*)
	PWM_Y26_SET:UINT;
	PWM_Y13:UINT;  (*A79 动力头正转Y13*)
	PWM_Y13_SET:UINT;
	PWM_Y14:UINT;  (*A80 动力头反转Y14*)
	PWM_Y14_SET:UINT;	
	PWM_Y21:UINT;  (*A81 左回转Y21*)
	PWM_Y21_SET:UINT;	
		
	(*B端口*)
	
	(***********输如************)
	AI_P8:UINT;    (*B06 回转制动压力P8*)
(*	AI_:UINT;  (*B36 蓄能器油压*)
	AI_:UINT;  (*B37 蓄能器气压*)
	AI_:UINT;      (*B38 主卷马达M1压力*)
	AI_:UINT;      (*B39 主卷马达M2压力*)
	(在GVL_SaveEngine中声明)
*)	
	
	(*PI*)
	PI_Q1:UINT;(*B44 泵1流量*)
	PI_Q1Freq:REAL;(*B44 泵1流量*)
	PI_Q2Freq:REAL;(*B45 泵2流量*)
	PI_Q2:UINT;(*B45 泵2流量*)
	PI_QAc:UINT;(*B46 蓄能器流量*)
	PI_QAcFreq:REAL;(*B46 蓄能器流量*)
	PI_QM1:UINT;(*B47 马达上升入口流量*)
	PI_QM1Freq:REAL;(*B47 马达上升入口流量*)
	(***********输出************)
	(*PWM*)
	PWM_Y22:UINT;  (*B16 右回转Y22*)
	PWM_Y22_SET:UINT;
	PWM_Y27:UINT;  (*B17 立桅左油缸伸Y27*)
	PWM_Y27_SET:UINT;	
	  				(*B18 备用*)
	
	PWM_Y28:UINT;  (*B19 立桅左油缸缩Y28*)
	PWM_Y28_SET:UINT;	
					  (*B20 备用*)
					  
	PWM_Y29:UINT;  (*B21 立桅右油缸伸Y29*)
	PWM_Y29_SET:UINT;	
	PWM_Y60:UINT;  (*B22 动力头3_1正转Y60*)
	PWM_Y60_SET:UINT;	
	PWM_Y61:UINT;  (*B23 动力头3_1反转Y61*)
	PWM_Y61_SET:UINT;	
	PWM_Y39:UINT;  (*B24 泵1建压Y39*)
	PWM_Y39_SET:UINT;
	PWM_Y31:UINT;  (*B63 支腿油缸伸Y31*)
	PWM_Y31_SET:UINT;	
	PWM_Y30:UINT;  (*B64 立桅右油缸缩Y30*)
	PWM_Y30_SET:UINT;	
	PWM_Y32:UINT;  (*B65 支腿油缸缩Y32*)
	PWM_Y32_SET:UINT;	
	PWM_Y35:UINT;	
	(*PWM_Y35:UINT;  (*B66 延时断电*)
	PWM_Y35_SET:UINT;	*)
	DOH_YS3:BOOL;(*B66 延时断电 实际为Y72*)
	PWM_Y41:UINT;  (*B67  动力头快速回油（反转）Y41*)
	PWM_Y41_SET:UINT;	
	(*DOH_Y58:BOOL;  (*B68 加压快电磁阀Y58*)*)
	DOH_Y58:BOOL;
	DOH_Y64:BOOL; (*B68 主卷限制Y64*)
	PWM_Y40:UINT;  (*B69 泵2建压Y40*)	
	PWM_Y40_SET:UINT;	
	PWM_Y42:UINT;  (*B70  动力头快速回油（正转）Y42*)
	PWM_Y42_SET:UINT;		
	PWM_Y34:UINT;  (*B73  动力头变量*)
	PWM_Y34_SET:UINT;
	PWM_Y37:UINT;  (*B74 直线行走使能Y37*)
	PWM_Y37_SET:UINT;			
	PWM_Y46:UINT;  (*B75  涨紧伸Y46*)
	PWM_Y46_SET:UINT;
	PWM_Y38:UINT;  (*B76 备用*)
	PWM_Y38_SET:UINT;			
	PWM_Y49:UINT;  (*B77  冷却泵变量控制Y49*)
	PWM_Y49_SET:UINT;			
	PWM_Y63:UINT;  (*B78  加压调节Y63*)
	PWM_Y63_SET:UINT;			
	
	PWM_Y59:UINT;  (*B80  动力头正转合流（正转）Y59*)
	PWM_Y59_SET:UINT;	
	
	
		
	
	
	(*DOH*)
	DOH_Y72:BOOL;    (*B66 Y72*)	
	DOH_Y71:BOOL;    (*B76 Y71*)
	
	
	(*IO模块*)
	(*DOH*)
	DOH_Y50:BOOL;  (*IO1 回转开锁Y50*)
	DOH_Y51:BOOL;  (*IO2 先导电磁阀Y51*)
	DOH_Y52:BOOL;  (*IO3 绳涨紧/鹅头油缸切换Y52*) 
	DOH_Y53:BOOL;  (*IO4 履带/支腿切换Y53*)
	DOH_Y54:BOOL;  (*IO5 支腿/鹅头油缸切换*)
	DOH_Y55:BOOL;  (*IO6 主卷开锁*)
	DOH_Y56:BOOL;  (*IO7 主卷浮动*)
	DOH_Y57:BOOL;  (*IO10 冷却风扇溢流阀*)
	DOH_Y59:BOOL;  (*IO11 动力头正转回油*)
	DOH_JK1:BOOL;  (*IO12 监控1*)
	DOH_JK2:BOOL;  (*IO13 监控2*)
	DOH_JK3:BOOL;  (*IO14 监控3*)
	DOH_JK4:BOOL;  (*IO15 监控4*)
	DOH_70:BOOL;   (*IO18 警示灯报警1*)
	DOH_73:BOOL;   (*IO19 警示灯报警2*)
	DOH_B1:BOOL;   (*IO20 蜂鸣器*)

END_VAR

// StandardPLC/Application/GLV/CAN_GVL
VAR_GLOBAL
(****发送数据****)
(************发送到显示屏数据**************)
	CANO_MainPUMP_Press1:UINT;
	CANO_MainPUMP_Press2:UINT;
	CANO_Fubeng_Press:UINT;
	CANO_SensorError_MainPUMP1Press:BOOL;
	CANO_SensorError_MainPUMP2Press:BOOL;
	CANO_SensorError_FubengPress:BOOL;
(*主界面数据*)
	DO_Begin_on:BOOL;
(*187*)
	CANO_ANGLE_X:UINT;
	CANO_ANGLE_Y:UINT;
	CANO_R_ANGLE:UINT;
	CANO_Hyd_Tem:UINT;
(*287*)

	CANO_water_tem:INT;
	CANO_JiayaPressure:UINT;
(*387*)

	CANO_DEPTH:UINT;
	CANO_FUEL_LEVEL:UINT;
	CANO_SPEED:UINT;
(*487*)
(*byte0*)
	CANO_TooLow_BatteryVol:BOOL;
	CANO_RotationModle:BOOL;(*回转模式1自动，0手动*)
	CANO_TooLow_FUEL_LEVEL:BOOL;
	CANO_UpLimitWarn: BOOL;
(*byte1*)
	CANO_TooHigh_HydOilTem:BOOL;
	CANO_TooLow_OilPress:BOOL;
	CANO_TooHigh_WaterTem:BOOL;
	CANO_LevelModle:BOOL;(*调平模式 1自动，0手动*)	
	CANO_Limite_Cancel:BOOL;

	CANO_DonglitouPressure:UINT;
	CANO_ZhuJuanPressure:UINT;
	CANO_Lub_Press:UINT;
(*288*)
(*byte0*)
	CANO_SensorError_Joy:BOOL;
	CANO_SensorError_Angle:BOOL;
	CANO_SensorError_Rotation:BOOL;
	CANO_SensorError_DonglitouPress:BOOL;
	CANO_SensorError_JiaYaPress:BOOL;
	CANO_SensorError_HydOilTem:BOOL;
	CANO_SensorError_ZhuJuanPress:BOOL;
(*byte1*)
	CANO_SensorError_FuelLevel:BOOL;
	CANO_SensorError_Depth:BOOL;
	CANO_SensorError_GPScan:BOOL;
	CANO_SensorError_PAtomsPre:BOOL;//蓄能器气压
	CANO_SensorError_PAcPre:BOOL;//蓄能器油压
	CANO_SensorError_PM1:BOOL;
	CANO_SensorError_PM2:BOOL;

(*388*)
(*byte0*)
(*byte1*)
	CANO_PowerHeadTorque: UINT;
(*488*)
	CANO_VOL_VALUE:UINT;
	CANO_PowerHeadSpeed: UINT;

(*189*)

(*289*)

	CANO_engine_hour_h:DINT;
(*389*)

(*489*)
	CANO_Accumu_Fuel:UDINT;
(*18A*)

	CANO_ACCMUDEPTH:UDINT;
	CANO_LimiteModle:USINT;
	CANO_engine_hour_m:BYTE;
(*28A*)
(*38A*)
(*48A*)
(*18B*)
(*28B*)
(*38B*)
(*48B*)

(*18C*)
	CANO_RotationStop_Pressure: UINT;
(*28C*)
	CANO_PilotPressure:UINT;
(*38C*)
	Codes_SPN_1:UDINT;
	Codes_SPN_2:UDINT;
(*48C*)
	Codes_SPN_3:UDINT;
	Codes_SPN_4:UDINT;
(*18D*)
	CANO_AO_Y23:UINT;					(*12_E*)(*OUT06_E M4阀*)
(*38D*)
	CANO_AO_Y22:UINT;					(*13_E*)(*OUT05_E M4阀*)
	CANO_AO_Y21:UINT;					(*14_E*)(*OUT04_E M4阀*)
(*48D*)
	Codes_SPN_5:UDINT;
	Codes_SPN_6:UDINT;
(*186*)
	Codes_SPN_7:UDINT;
	Codes_SPN_8:UDINT;
(*286*)
	Codes_SPN_9:UDINT;
	Codes_SPN_10:UDINT;
(*386*)
	Codes_FMI_1:BYTE;
	Codes_FMI_2:BYTE;
	Codes_FMI_3:BYTE;
	Codes_FMI_4:BYTE;
	Codes_FMI_5:BYTE;
	Codes_FMI_6:BYTE;
	Codes_FMI_7:BYTE;
	Codes_FMI_8:BYTE;
(*486*)
	Codes_FMI_9:BYTE;
	Codes_FMI_10:BYTE;
(*byte2*)
	CANO_SensorError_Tension:BOOL;
	CANO_SensorError_PoiltPress:BOOL;

	CANO_ChuDiBaohu: BOOL;
	CANO_DaiGan_Warn: BOOL;


(*185*)
	
(*285*)
	CANO_PLC_Hardward_Versions:UINT;
	CANO_PLC_Software_Versions:UINT;
	CANO_GPS_Hardward_Versions:UINT;
	CANO_GPS_Software_Versions:UINT;
(*385*)

(*784*)
	CANO_MainWinchTension:UINT;
	CANO_LoadRate:UINT;
	CANO_RotationPress:UINT;
(*18D*)
	MainWinch_Speed: INT;
	CANO_MainWinch_Speed: UINT;
(*CFA*)
	CANO_CFA_Flow:UINT;
	CANO_CFA_Press:UINT;
	CANO_MainWinchSpeed:UINT;
(*发动机数据*)
	Codes_all :BYTE;
	Codes_SPN :ARRAY[1..10] OF  UDINT;
    Codes_FMI :ARRAY[1..10] OF  BYTE;
	
	CANO_LastDepth:UINT;
(*GPS*)
	CAN_GPS_STATUS_UnLock						:BOOL;
	CAN_GpsTempUnlockDoing						:BOOL;
	CAN_NewGpsRecLockCommand				:UINT;
	CAN_NewGpsRecUnLockCommand			:UINT;
	CAN_TranData_NewGps1						:UINT;
	CAN_TranData_NewGps2						:UINT;
    GpsPasswordTempUnlockCount 				:UINT;
	GPS_Controller_Lock: BOOL;
	GPS_Relay_Lock: BOOL;
	GPS_Delay_Lock: BOOL;
	GPS_Remove_Lock: BOOL;
	GPS_Cover_Lock: BOOL;
	GPS_Controller_UnLock: BOOL;
	GPS_Relay_UnLock: BOOL;
	GPS_Delay_UnLock: BOOL;
	GPS_Remove_UnLock: BOOL;
	GPS_Cover_UnLock: BOOL;
	GPS_Temp: UINT;
	GPS_Linshi_Password: UINT;
	CanNewGpsRealFakeTargetData: UINT;
	GPS_CanNewGpsRealFakeRecData: UINT;
	CanNewGpsRealFakeResult:BOOL;
	Controller_STATUS : BOOL;
	Relay_STATUS : BOOL;
	Delay_STATUS : BOOL;
	Remove_STATUS: BOOL;
	Cover_STATUS: BOOL;
	GPS_NUM:BYTE;
	CAN_GPS_STATUS1:BOOL;
(**)
	DI_LHandle_SB1:BOOL;		(* 左手柄按钮1*)
	DI_LHandle_SB2:BOOL;		(* 左手柄按钮2*)
	DI_LHandle_SB3:BOOL;		(* 左手柄按钮3*)
	DI_LHandle_SB4:BOOL;		(*左手柄按钮4*)
	DI_LHandle_SB5:BOOL;		(*左手柄按钮5*)
	DI_LHandle_SB6:BOOL;		(*左手柄按钮6*)
	DI_LHandle_Enable:BOOL:=TRUE;
	DI_LHandle_SB7: BOOL;(*背部按钮*)

	DI_RHandle_SB1:BOOL;		(*右手柄按钮1*)
	DI_RHandle_SB2:BOOL;		(*右手柄按钮2*)
	DI_RHandle_SB3:BOOL;		(*右手柄按钮3*)
	DI_RHandle_SB4:BOOL;		(*右手柄按钮4*)
	DI_RHandle_SB5:BOOL;		(*右手柄按钮5*)
	DI_RHandle_SB6:BOOL;		(*右手柄按钮6*)
	DI_RHandle_Enable:BOOL:=TRUE;
	DI_RHandle_SB7:BOOL;
	
(****接收数据****)
(****接收数据****)
(*显示屏接收参数*)
(*主界面*)
	CANI_Button_RotationOriginal:BOOL:=FALSE;
	CANI_Button_DepthClear:BOOL:=FALSE;
	CANI_Button_BuzzSwitch:BOOL:=FALSE;
	CANI_Button_FloatSwitch:BOOL:=FALSE;
(*调平界面*)
	CANI_Button_LEVER_Auto:BOOL:=FALSE;
	CANI_Button_LEVER_XPlus:BOOL:=FALSE;
	CANI_Button_LEVER_XSubtract:BOOL:=FALSE;
	CANI_Button_LEVER_YPlus:BOOL:=FALSE;
	CANI_Button_LEVER_YSubtract:BOOL:=FALSE;
	CANI_Button_LEVER_Manual:BOOL:=FALSE;
(*调试界面*)
	CANI_Button_Debug_LStretchOut:BOOL:=FALSE;
	CANI_Button_Debug_LRetraction:BOOL:=FALSE;
	CANI_Button_Debug_RStretchOut:BOOL:=FALSE;
	CANI_Button_Debug_RRetraction:BOOL:=FALSE;
(*记录清零界面*)
	CANI_Button_RecordClear:BOOL:=FALSE;
	CANI_Button_RecordClear1:BOOL:=FALSE;
(*主参数*)
	CANI_Button_MainSetting_XZero:BOOL:=FALSE;
	CANI_Button_MainSetting_YZero:BOOL:=FALSE;
(*桅杆标定界面*)
	CANI_Button_L_Limit:BOOL:=FALSE;
	CANI_Button_R_Limit:BOOL:=FALSE;
(*油门设置界面*)
	CANI_Button_YouMen_Min:BOOL:=FALSE;
	CANI_Button_YouMen_Max:BOOL:=FALSE;
	CANI_Button_YouMen_Motor:BOOL:=FALSE;
(*加压卷扬设置界面*)
	CANI_Button_JiYaWinchDepth_Clear:BOOL:=FALSE;
	DoLiTou_Location_clear:BOOL:=FALSE;
(*****薄膜按键*****)
	CANI_WorkModeSwitch:BOOL;(*调整作业开关*)
	CANI_MaiWinFloatSwitch:BOOL;(*主卷浮动开关*)
	CANI_ColdFunSwitch:BOOL;(*冷却开关*)
	CANI_DonglitouHSwitch:BOOL;(*动力头重载模式*)
	CANI_DonglitouLSwitch:BOOL;(*动力头轻载模式*)
	CANI_DonglitouMSwitch:BOOL;(*动力头中载模式*)
	CANI_IdleEnbleSwitch:BOOL;(*自动怠速开关*)
	CANI_DongLiTouPressLimitSwitch:BOOL;(*加压限压开关*)
	CANI_DonglitouADDSwitch:BOOL;(*动力头转速增加开关*)
	CANI_DonglitouSUBSwitch:BOOL;(*动力头转速减小开关*)
	CANI_MoShiSwitch:BOOL;(*模式开关*)
	CANI_CFASwitch:BOOL;(*CFA开关*)
	CANI_RotationSuoSwitch:BOOL;(*回转制动油缸缩开关*)
	CANI_RotationShenSwitch:BOOL;(*回转制动油缸伸开关*)
	CANI_ShengZhangJinSwitch:BOOL;(*绳张紧开关*)
	CANI_LvDaiShenSuoSwitch:BOOL;(*履带伸缩开关*)
	CANI_ETouYouGangSwitch:BOOL;(*鹅头油缸开关*)
	CANI_MidSpeedSwitch:BOOL;(*发动机中速开关*)
	CANI_JiaYaFastSwitch:BOOL;(*加压快开关*)
	CANI_DongLiTouLimiSwitcht:BOOL;(*动力头限扭*)
	CANI_ECOSwitch: BOOL;(*ECO模式开关*)
	CANI_FuZhuRunhuaSwitch:BOOL;(*辅助润滑*)
	CANI_DongLiTouSpeedSlowSwitch:BOOL;(*动力头慢速*)
	CANI_DongLiTouAutoSwitch: BOOL;(*动力头回转锁定*)

	AI_ANGLE_X   :UINT;      (*采用CAN总线倾CAN总线读入*)
	AI_ANGLE_Y  :UINT;       (*采用CAN总线倾角传感器，从CAN总线读入*)
	(* 倾角传感器零位设置*)
	CANI_Button_Zero_AngleY:BOOL;
	CANI_Button_Zero_AngleX:BOOL;
	PAR_FUEL_LEVER_MINLABEL:UINT;
	PAR_FUEL_LEVER_MAXLABEL:UINT;
	PAR_FUEL_LEVER_ALARMLABEL:UINT;
(*左右手柄数据*)
	CANI_JOYX_L:UINT:=2500;
	CANI_JOYY_L:UINT:=2500;
	CANI_JOYX_R:UINT:=2500;
	CANI_JOYY_R:UINT:=2500;
	CANI_JOY_SB1:BOOL;
	CANI_JOY_SB2:BOOL;
	CANI_JOY_SB3:BOOL;
	CANI_JOY_SB4:BOOL;
	CANI_JOY_SB5:BOOL;
	CANI_JOY_SB6:BOOL;
	CANI_JOY_SB7:BOOL;
	CANI_JOY_SB8:BOOL;
	CANI_JOY_SB9:BOOL;
	CANI_JOY_SB10:BOOL;
	DI_RHandle_SB8A: BOOL;
	DI_RHandle_SB8B: BOOL;
	DI_LHandle_SB4_UINT: USINT;
	DI_RHandle_SB7_UINT: USINT;
(*脚踏板数据*)
	CANI_JOY_Jiao_L:UINT:=2500;
	CANI_JOY_Jiao_R:UINT:=2500;
(********)
	JOYX_L:UINT;
	JOYY_L:UINT;
	JOYX_R:UINT;
	JOYY_R:UINT;
	JOY_Jiao_L:UINT;
	JOY_Jiao_R:UINT;

	PWM_JOYX_L_UP: UINT;
	PWM_JOYX_L_DOWN: UINT;
	PWM_JOYY_L_UP: UINT;
	PWM_JOYY_L_DOWN: UINT;

	PWM_JOYX_R_UP: UINT;
	PWM_JOYX_R_DOWN: UINT;
	PWM_JOYY_R_UP: UINT;
	PWM_JOYY_R_DOWN: UINT;

	PWM_JOY_Jiao_L_UP: UINT;
	PWM_JOY_Jiao_L_DOWN: UINT;
	PWM_JOY_Jiao_R_UP: UINT;
	PWM_JOY_Jiao_R_DOWN: UINT;
	

	AI_ECM2_Flag: UINT;
END_VAR

// SafetyPLC/Application/EVL
(* THIS EVL IS AUTOGENERATED. DO NOT MODIFY THESE ATTRIBUTES. *)
{attribute 'location' := '16#800' }
{attribute 'linkalways'}
{attribute 'qualified_only'}
VAR_GLOBAL

END_VAR

// StandardPLC/Application/PLC_PRG
PROGRAM PLC_PRG
VAR
	ZONGXIAN: ZONGXIANJISUAN;
	sensor_x:UINT;
	sensor_y:UINT;
	censor: censor_cali;
	CAN_XY: CAN_XY;
	ANGLE_X: INT;
	ANGLE_Y: INT;
	MODE_ROTATE:MODE_ROTATE;
	ROTATEAUTO:ROTATE_AUTO;
	
	MODE_ROTATE_AU: BOOL;
	MODE_ROTATE_MA: BOOL;
	IncEncoder_0: ifmFastInput.IncEncoder;
	ttt:real;
END_VAR

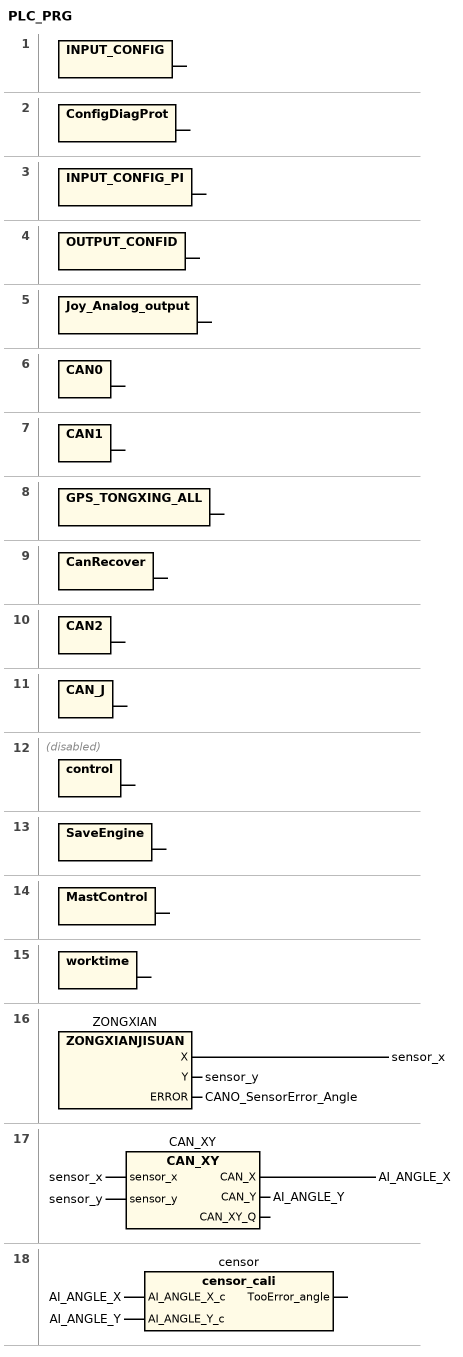
// NETWORK 1
INPUT_CONFIG();

// NETWORK 2
ConfigDiagProt();

// NETWORK 3
INPUT_CONFIG_PI();

// NETWORK 4
OUTPUT_CONFID();

// NETWORK 5
Joy_Analog_output();

// NETWORK 6
CAN0();

// NETWORK 7
CAN1();

// NETWORK 8
GPS_TONGXING_ALL();

// NETWORK 9
CanRecover();

// NETWORK 10
CAN2();

// NETWORK 11
CAN_J();

// NETWORK 12 (disabled)
// control();

// NETWORK 13
SaveEngine();

// NETWORK 14
MastControl();

// NETWORK 15
worktime();

// NETWORK 16
ZONGXIAN(Y => sensor_y, ERROR => CANO_SensorError_Angle); // ZONGXIANJISUAN
sensor_x := ZONGXIAN.X;

// NETWORK 17
CAN_XY(sensor_x := sensor_x, sensor_y := sensor_y, CAN_Y => AI_ANGLE_Y);
AI_ANGLE_X := CAN_XY.CAN_X;

// NETWORK 18
censor(AI_ANGLE_X_c := AI_ANGLE_X, AI_ANGLE_Y_c := AI_ANGLE_Y); // censor_cali

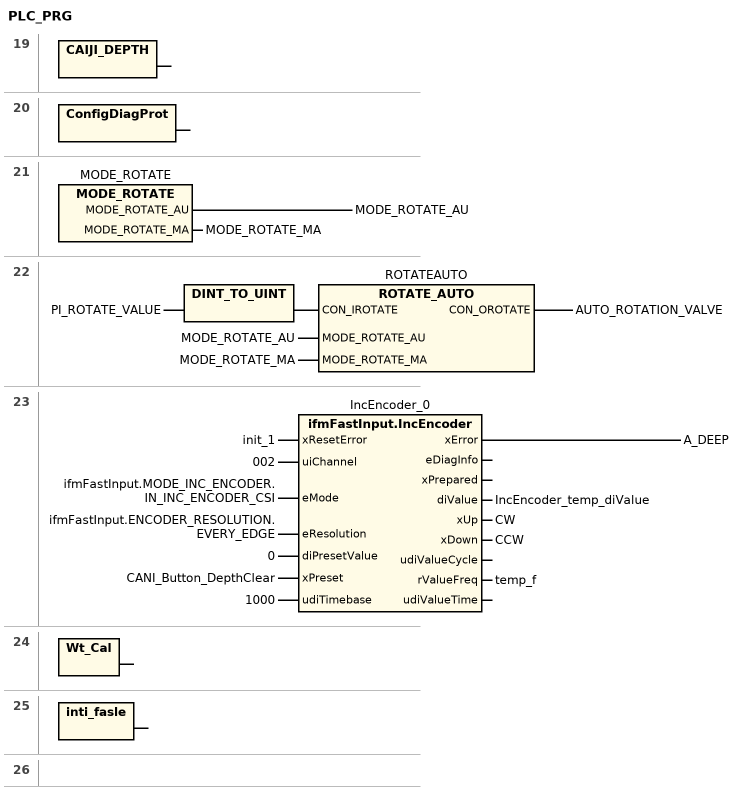
// NETWORK 19
CAIJI_DEPTH();

// NETWORK 20
ConfigDiagProt();

// NETWORK 21
MODE_ROTATE(MODE_ROTATE_MA => MODE_ROTATE_MA);
MODE_ROTATE_AU := MODE_ROTATE.MODE_ROTATE_AU;

// NETWORK 22
ROTATEAUTO(
    CON_IROTATE := DINT_TO_UINT(PI_ROTATE_VALUE),
    MODE_ROTATE_AU := MODE_ROTATE_AU,
    MODE_ROTATE_MA := MODE_ROTATE_MA); // ROTATE_AUTO
AUTO_ROTATION_VALVE := ROTATEAUTO.CON_OROTATE;

// NETWORK 23
IncEncoder_0(
    xResetError := init_1,
    uiChannel := 002,
    eMode := ifmFastInput.MODE_INC_ENCODER.IN_INC_ENCODER_CSI,
    eResolution := ifmFastInput.ENCODER_RESOLUTION.EVERY_EDGE,
    diPresetValue := 0,
    xPreset := CANI_Button_DepthClear,
    udiTimebase := 1000,
    diValue => IncEncoder_temp_diValue,
    xUp => CW,
    xDown => CCW,
    rValueFreq => temp_f); // ifmFastInput.IncEncoder
A_DEEP := IncEncoder_0.xError;

// NETWORK 24
Wt_Cal();

// NETWORK 25
inti_fasle();

// NETWORK 26

END_PROGRAM

// StandardPLC/Application/IO_CONFIG/INPUT_CONFIG
PROGRAM INPUT_CONFIG
VAR
	(*脉冲输入点*)
	INPUT_A25:ifmIOcommon.Input;
	INPUT_A26:ifmIOcommon.Input;
	
	(* DIH *)	
	INPUT_A27:ifmIOcommon.Input;
	INPUT_A28:ifmIOcommon.Input;
	INPUT_A36:ifmIOcommon.Input;
	INPUT_A37:ifmIOcommon.Input;
	INPUT_A38:ifmIOcommon.Input;
	INPUT_A39:ifmIOcommon.Input;
	INPUT_A44:ifmIOcommon.Input;
	INPUT_A45:ifmIOcommon.Input;
	INPUT_A46:ifmIOcommon.Input;
	INPUT_A47:ifmIOcommon.Input;
	INPUT_B6:ifmIOcommon.Input;
	INPUT_B10:ifmIOcommon.Input;
	
	
	(* DIL *)
	INPUT_A40:ifmIOcommon.Input;
	INPUT_A41:ifmIOcommon.Input;
	INPUT_A42:ifmIOcommon.Input;
	INPUT_A43:ifmIOcommon.Input;
	
	(* AI *)
	INPUT_A55:ifmIOcommon.Input;
	INPUT_A56:ifmIOcommon.Input;
	INPUT_A57:ifmIOcommon.Input;
	INPUT_A58:ifmIOcommon.Input;
	INPUT_A59:ifmIOcommon.Input;
	INPUT_A60:ifmIOcommon.Input;
	INPUT_A61:ifmIOcommon.Input;
	INPUT_A62:ifmIOcommon.Input;
	INPUT_A63:ifmIOcommon.Input;
	INPUT_A64:ifmIOcommon.Input;
	INPUT_A65:ifmIOcommon.Input;
	INPUT_A66:ifmIOcommon.Input;
	INPUT_A67:ifmIOcommon.Input;
	INPUT_A68:ifmIOcommon.Input;
	INPUT_A69:ifmIOcommon.Input;
	INPUT_A70:ifmIOcommon.Input;
	INPUT_B36:ifmIOcommon.Input;//节能蓄能器油压
	INPUT_B07:ifmIOcommon.Input;//节能蓄能器气压
	INPUT_B38:ifmIOcommon.Input;//节能M1压力下放马达出口
	INPUT_B39:ifmIOcommon.Input;//节能M2压力下放马达入口
	INPUT_B44:ifmFastInput.Period;//PI_Q1
	INPUT_B45:ifmFastInput.Period;//PI_Q2
	INPUT_B46:ifmFastInput.Period;//PI_QAc
	INPUT_B47:ifmFastInput.Period;//PI_QM1 上升入口
	
	AI_SQ1_ZhongJian:UINT;
	AI_SQ2_ZhongJian:UINT;
	
	INPUT_B57:ifmIOcommon.Input;
	
	
END_VAR

(*PI*)

(* DIH *)
(*INPUT_A27(            (* IN0002深度接近开关SQ1 *)
	xResetError:= init_1, 
	uiChannel:= 002, 
	eMode:=ifmIOcommon.MODE_INPUT.IN_DIGITAL_CSI, 
	eFilter:=ifmIOcommon.FILTER_INPUT.UNCHANGED, 
	xError=> , 
	eDiagInfo=> , 
	xPrepared=> , 
	xValueDigital=> DIH_SQ1, 
	uiValueAnalogue=> );
	
	
INPUT_A28(            (* IN0003深度接近开关SQ2 *)
	xResetError:= init_1, 
	uiChannel:= 003, 
	eMode:=ifmIOcommon.MODE_INPUT.IN_DIGITAL_CSI, 
	eFilter:=ifmIOcommon.FILTER_INPUT.UNCHANGED, 
	xError=> , 
	eDiagInfo=> , 
	xPrepared=> , 
	xValueDigital=> DIH_SQ2, 
	uiValueAnalogue=> );*)
		
INPUT_A36(            (* IN0800 电手柄按钮JOY *)
	xResetError:= init_1, 
	uiChannel:= 800, 
	eMode:=ifmIOcommon.MODE_INPUT.IN_DIGITAL_CSI, 
	eFilter:=ifmIOcommon.FILTER_INPUT.FILTER_2, 
	xError=> , 
	eDiagInfo=> , 
	xPrepared=> , 
	xValueDigital=> DIH_JOY, 
	uiValueAnalogue=> );
	
INPUT_A37(            (* IN0801 浮动脚踏开关SA8 *)
	xResetError:= init_1, 
	uiChannel:= 801, 
	eMode:=ifmIOcommon.MODE_INPUT.IN_DIGITAL_CSI, 
	eFilter:=ifmIOcommon.FILTER_INPUT.FILTER_2, 
	xError=> , 
	eDiagInfo=> , 
	xPrepared=> , 
	xValueDigital=> DIH_SA8, 
	uiValueAnalogue=> );	
	
INPUT_A38(            (* IN0802 回油滤芯开关SP4 *)
	xResetError:= init_1, 
	uiChannel:= 802, 
	eMode:=ifmIOcommon.MODE_INPUT.IN_DIGITAL_CSI, 
	eFilter:=ifmIOcommon.FILTER_INPUT.FILTER_2, 
	xError=> , 
	eDiagInfo=> , 
	xPrepared=> , 
	xValueDigital=> DIH_SP4, 
	uiValueAnalogue=> );
		
INPUT_A39(            (* IN0900 平举下限位 SQ12 *)
	xResetError:= init_1, 
	uiChannel:= 900, 
	eMode:=ifmIOcommon.MODE_INPUT.IN_DIGITAL_CSI, 
	eFilter:=ifmIOcommon.FILTER_INPUT.FILTER_2, 
	xError=> , 
	eDiagInfo=> , 
	xPrepared=> , 
	xValueDigital=> DIH_SQ12, 
	uiValueAnalogue=> );	
		
INPUT_A44(            (* IN0300 桅杆左限位开关 SQ5 *)
	xResetError:= init_1, 
	uiChannel:= 300, 
	eMode:=ifmIOcommon.MODE_INPUT.IN_DIGITAL_CSI, 
	eFilter:=ifmIOcommon.FILTER_INPUT.FILTER_2, 
	xError=> , 
	eDiagInfo=> , 
	xPrepared=> , 
	xValueDigital=> DIH_SQ5, 
	uiValueAnalogue=> );		
		
INPUT_A45(            (* IN0301 桅杆右限位开关 SQ6 *)
	xResetError:= init_1, 
	uiChannel:= 301, 
	eMode:=ifmIOcommon.MODE_INPUT.IN_DIGITAL_CSI, 
	eFilter:=ifmIOcommon.FILTER_INPUT.FILTER_2, 
	xError=> , 
	eDiagInfo=> , 
	xPrepared=> , 
	xValueDigital=> DIH_SQ6, 
	uiValueAnalogue=> );	
	
INPUT_A47(            (* IN0401 动力头慢速 SA18 *)
	xResetError:= init_1, 
	uiChannel:= 401, 
	eMode:=ifmIOcommon.MODE_INPUT.IN_DIGITAL_CSI, 
	eFilter:=ifmIOcommon.FILTER_INPUT.FILTER_2, 
	xError=> , 
	eDiagInfo=> , 
	xPrepared=> , 
	xValueDigital=> DIH_SA18, 
	uiValueAnalogue=> );	
	
INPUT_A70(            (* IN0203 行走快速SA19 *)
	xResetError:= init_1, 
	uiChannel:= 203, 
	eMode:=ifmIOcommon.MODE_INPUT.IN_DIGITAL_CSI, 
	eFilter:=ifmIOcommon.FILTER_INPUT.FILTER_2, 
	xError=> , 
	eDiagInfo=> , 
	xPrepared=> , 
	xValueDigital=> DIH_SA19, 
	uiValueAnalogue=> );	
	
INPUT_B10(            (* IN1200 钥匙开关3*)
	xResetError:= init_1, 
	uiChannel:= 1200, 
	eMode:=ifmIOcommon.MODE_INPUT.IN_DIGITAL_CSI, 
	eFilter:=ifmIOcommon.FILTER_INPUT.FILTER_2, 
	xError=> , 
	eDiagInfo=> , 
	xPrepared=> , 
	xValueDigital=> DIH_power3, 
	uiValueAnalogue=> );	
	
INPUT_B6(            (* IN1100 动力头限制扭矩SA15*)
	xResetError:= init_1, 
	uiChannel:= 1100, 
	eMode:=ifmIOcommon.MODE_INPUT.IN_DIGITAL_CSI, 
	eFilter:=ifmIOcommon.FILTER_INPUT.FILTER_2, 
	xError=> , 
	eDiagInfo=> , 
	xPrepared=> , 
	xValueDigital=> DIH_SA15, 
	uiValueAnalogue=> );	
(*DIL*)	
INPUT_A40(            (* IN0500 先导开关 SQ3 *)
	xResetError:= init_1, 
	uiChannel:= 500, 
	eMode:=ifmIOcommon.MODE_INPUT.IN_DIGITAL_CSO, 
	eFilter:=ifmIOcommon.FILTER_INPUT.FILTER_2, 
	xError=> , 
	eDiagInfo=> , 
	xPrepared=> , 
	xValueDigital=> DIL_SQ3, 
	uiValueAnalogue=> );	

INPUT_A41(            (* IN0501 主卷上限位 SQ4 *)
	xResetError:= init_1, 
	uiChannel:= 501, 
	eMode:=ifmIOcommon.MODE_INPUT.IN_DIGITAL_CSO, 
	eFilter:=ifmIOcommon.FILTER_INPUT.FILTER_2, 
	xError=> , 
	eDiagInfo=> , 
	xPrepared=> , 
	xValueDigital=> DIL_SQ4, 
	uiValueAnalogue=> );
	
INPUT_A42(            (* IN0502 主卷上限位 SQ11*)
	xResetError:= init_1, 
	uiChannel:= 502, 
	eMode:=ifmIOcommon.MODE_INPUT.IN_DIGITAL_CSO, 
	eFilter:=ifmIOcommon.FILTER_INPUT.FILTER_2, 
	xError=> , 
	eDiagInfo=> , 
	xPrepared=> , 
	xValueDigital=> DIL_SQ11, 
	uiValueAnalogue=> );	
	
INPUT_A43(            (* IN0503 液位传感器 SQ13*)
	xResetError:= init_1, 
	uiChannel:= 503, 
	eMode:=ifmIOcommon.MODE_INPUT.IN_DIGITAL_CSO, 
	eFilter:=ifmIOcommon.FILTER_INPUT.FILTER_2, 
	xError=> , 
	eDiagInfo=> , 
	xPrepared=> , 
	xValueDigital=> DIL_SQ13, 
	uiValueAnalogue=> );	
	
(*AI*)
INPUT_A55(            (* IN0600 加压压力P1*)
	xResetError:= init_1, 
	uiChannel:= 600, 
	eMode:=ifmIOcommon.MODE_INPUT.IN_CURRENT_CSI, 
	eFilter:=ifmIOcommon.FILTER_INPUT.FILTER_2, 
	xError=> , 
	eDiagInfo=> , 
	xPrepared=> , 
	xValueDigital=> , 
	uiValueAnalogue=> AI_P1 );
	
INPUT_A56(            (* IN0601 动力头压力P2*)
	xResetError:= init_1, 
	uiChannel:= 601, 
	eMode:=ifmIOcommon.MODE_INPUT.IN_CURRENT_CSI, 
	eFilter:=ifmIOcommon.FILTER_INPUT.FILTER_2, 
	xError=> , 
	eDiagInfo=> , 
	xPrepared=> , 
	xValueDigital=> , 
	uiValueAnalogue=> AI_P2);		
	
INPUT_A57(            (* IN0602 主卷压力P3*)
	xResetError:= init_1, 
	uiChannel:= 602, 
	eMode:=ifmIOcommon.MODE_INPUT.IN_CURRENT_CSI, 
	eFilter:=ifmIOcommon.FILTER_INPUT.FILTER_2, 
	xError=> , 
	eDiagInfo=> , 
	xPrepared=> , 
	xValueDigital=> , 
	uiValueAnalogue=> AI_P3);		
	
INPUT_A58(            (* IN0603 主泵1压力P11*)
	xResetError:= init_1, 
	uiChannel:= 603, 
	eMode:=ifmIOcommon.MODE_INPUT.IN_CURRENT_CSI, 
	eFilter:=ifmIOcommon.FILTER_INPUT.FILTER_2, 
	xError=> , 
	eDiagInfo=> , 
	xPrepared=> , 
	xValueDigital=> , 
	uiValueAnalogue=> AI_P11);		
	
INPUT_A59(            (* IN0700 主泵2压力P12*)
	xResetError:= init_1, 
	uiChannel:= 700, 
	eMode:=ifmIOcommon.MODE_INPUT.IN_CURRENT_CSI, 
	eFilter:=ifmIOcommon.FILTER_INPUT.FILTER_2, 
	xError=> , 
	eDiagInfo=> , 
	xPrepared=> , 
	xValueDigital=> , 
	uiValueAnalogue=> AI_P12);	
	
INPUT_A60(            (* IN0701 副泵/M4阀压力P6*)
	xResetError:= init_1, 
	uiChannel:= 701, 
	eMode:=ifmIOcommon.MODE_INPUT.IN_CURRENT_CSI, 
	eFilter:=ifmIOcommon.FILTER_INPUT.FILTER_4, 
	xError=> , 
	eDiagInfo=> , 
	xPrepared=> , 
	xValueDigital=> , 
	uiValueAnalogue=> AI_P6);		
	
INPUT_A61(            (* IN0702 先导压力P7*)
	xResetError:= init_1, 
	uiChannel:= 702, 
	eMode:=ifmIOcommon.MODE_INPUT.IN_CURRENT_CSI, 
	eFilter:=ifmIOcommon.FILTER_INPUT.FILTER_2, 
	xError=> , 
	eDiagInfo=> , 
	xPrepared=> , 
	xValueDigital=> , 
	uiValueAnalogue=> AI_P7);		
	
INPUT_A62(            (* IN0703 电手柄X轴 JOYX *)
	xResetError:= init_1, 
	uiChannel:= 703, 
	eMode:=ifmIOcommon.MODE_INPUT.IN_VOLTAGE_10, 
	eFilter:=ifmIOcommon.FILTER_INPUT.FILTER_2, 
	xError=> , 
	eDiagInfo=> , 
	xPrepared=> , 
	xValueDigital=> , 
	uiValueAnalogue=> AI_JOYX);		
	
INPUT_A63(            (* IN0100 电手柄Y轴 JOYY *)
	xResetError:= init_1, 
	uiChannel:= 100, 
	eMode:=ifmIOcommon.MODE_INPUT.IN_VOLTAGE_10, 
	eFilter:=ifmIOcommon.FILTER_INPUT.FILTER_2, 
	xError=> , 
	eDiagInfo=> , 
	xPrepared=> , 
	xValueDigital=> , 
	uiValueAnalogue=> AI_JOYY);		
	
INPUT_A64(            (* IN0101 燃油液位传感器 SP1 *)
	xResetError:= init_1, 
	uiChannel:= 101, 
	eMode:=ifmIOcommon.MODE_INPUT.IN_VOLTAGE_32, 
	eFilter:=ifmIOcommon.FILTER_INPUT.FILTER_2, 
	xError=> , 
	eDiagInfo=> , 
	xPrepared=> , 
	xValueDigital=> , 
	uiValueAnalogue=> AI_SP1);		
	
INPUT_A65(            (* IN0102 液压油温传感器 SP3 *)
	xResetError:= init_1, 
	uiChannel:= 102, 
	eMode:=ifmIOcommon.MODE_INPUT.IN_VOLTAGE_32, 
	eFilter:=ifmIOcommon.FILTER_INPUT.FILTER_2, 
	xError=> , 
	eDiagInfo=> , 
	xPrepared=> , 
	xValueDigital=> , 
	uiValueAnalogue=> AI_SP3);		
		
INPUT_A66(            (* IN0103 销轴传感器 SP7 *)
	xResetError:= init_1, 
	uiChannel:= 103, 
	eMode:=ifmIOcommon.MODE_INPUT.IN_CURRENT_CSI, 
	eFilter:=ifmIOcommon.FILTER_INPUT.FILTER_2, 
	xError=> , 
	eDiagInfo=> , 
	xPrepared=> , 
	xValueDigital=> , 
	uiValueAnalogue=> AI_SP7);	
	
INPUT_A67(            (* IN0200 左右倾角角度传感器 SP11 *)
	xResetError:= init_1, 
	uiChannel:= 200, 
	eMode:=ifmIOcommon.MODE_INPUT.IN_VOLTAGE_10, 
	eFilter:=ifmIOcommon.FILTER_INPUT.FILTER_2, 
	xError=> , 
	eDiagInfo=> , 
	xPrepared=> , 
	xValueDigital=> , 
	uiValueAnalogue=> AI_SP11);	
	
INPUT_A68(            (* IN0201 油门旋钮 ECM2/9 *)
	xResetError:= init_1, 
	uiChannel:= 201, 
	eMode:=ifmIOcommon.MODE_INPUT.IN_VOLTAGE_10, 
	eFilter:=ifmIOcommon.FILTER_INPUT.FILTER_2, 
	xError=> , 
	eDiagInfo=> , 
	xPrepared=> , 
	xValueDigital=> , 
	uiValueAnalogue=> AI_ECM2_9);		
	
INPUT_A69(            (* IN0202 加压压力P1A *)
	xResetError:= init_1, 
	uiChannel:= 202, 
	eMode:=ifmIOcommon.MODE_INPUT.IN_CURRENT_CSI, 
	eFilter:=ifmIOcommon.FILTER_INPUT.FILTER_4, 
	xError=> , 
	eDiagInfo=> , 
	xPrepared=> , 
	xValueDigital=> , 
	uiValueAnalogue=> AI_P1A);		
	


INPUT_B57(            (* IN1802 薄膜按键加压快按钮 *)
	xResetError:= init_1, 
	uiChannel:= 1802, 
	eMode:=ifmIOcommon.MODE_INPUT.IN_DIGITAL_CSI, 
	eFilter:=ifmIOcommon.FILTER_INPUT.FILTER_2, 
	xError=> , 
	eDiagInfo=> , 
	xPrepared=> , 
	xValueDigital=> CANI_JiaYaFastSwitch, 
	uiValueAnalogue=> );			
	
	(*节能增加输入*)
	
INPUT_B36(            (* IN1600 节能蓄能器油压*)
	xResetError:= init_1, 
	uiChannel:= 1600, 
	eMode:=ifmIOcommon.MODE_INPUT.IN_CURRENT_CSI, 
	eFilter:=ifmIOcommon.FILTER_INPUT.FILTER_2, 
	xError=> , 
	eDiagInfo=> , 
	xPrepared=> , 
	xValueDigital=> , 
	uiValueAnalogue=> GVL_SaveEngine.AI_PAcPreMv);
	
INPUT_B07(            (* IN1601 节能蓄能器气压*)
	xResetError:= init_1, 
	uiChannel:= 1101, 
	eMode:=ifmIOcommon.MODE_INPUT.IN_CURRENT_CSI, 
	eFilter:=ifmIOcommon.FILTER_INPUT.FILTER_2, 
	xError=> , 
	eDiagInfo=> , 
	xPrepared=> , 
	xValueDigital=> , 
	uiValueAnalogue=> GVL_SaveEngine.AI_PAtomsPreMv);	
		
INPUT_B38(            (* IN1602 节能M1压力*)
	xResetError:= init_1, 
	uiChannel:= 1602, 
	eMode:=ifmIOcommon.MODE_INPUT.IN_CURRENT_CSI, 
	eFilter:=ifmIOcommon.FILTER_INPUT.FILTER_2, 
	xError=> , 
	eDiagInfo=> , 
	xPrepared=> , 
	xValueDigital=> , 
	uiValueAnalogue=> GVL_SaveEngine.AI_PM1PreMv);

INPUT_B39(            (* IN1603 节能M2压力*)
	xResetError:= init_1, 
	uiChannel:= 1603, 
	eMode:=ifmIOcommon.MODE_INPUT.IN_CURRENT_CSI, 
	eFilter:=ifmIOcommon.FILTER_INPUT.FILTER_2, 
	xError=> , 
	eDiagInfo=> , 
	xPrepared=> , 
	xValueDigital=> , 
	uiValueAnalogue=> GVL_SaveEngine.AI_PM2PreMv);

END_PROGRAM

// StandardPLC/Application/IO_CONFIG/ConfigDiagProt
PROGRAM ConfigDiagProt
VAR
	DiagFunction_000:DiagFunction;
	DiagFunction_001:DiagFunction;
	DiagFunction_002:DiagFunction;
	DiagFunction_003:DiagFunction;
	DiagFunction_004:DiagFunction;
	DiagFunction_005:DiagFunction;
	DiagFunction_006:DiagFunction;
	DiagFunction_007:DiagFunction;
	DiagFunction_008:DiagFunction;
	
	DiagFunction_100:DiagFunction;
	DiagFunction_101:DiagFunction;
	DiagFunction_102:DiagFunction;
	DiagFunction_103:DiagFunction;
	DiagFunction_104:DiagFunction;
	DiagFunction_105:DiagFunction;
	DiagFunction_106:DiagFunction;
	DiagFunction_107:DiagFunction;
	DiagFunction_108:DiagFunction;
	
	DiagFunction_200:DiagFunction;
	DiagFunction_201:DiagFunction;
	DiagFunction_202:DiagFunction;
	DiagFunction_203:DiagFunction;
	DiagFunction_204:DiagFunction;
	DiagFunction_205:DiagFunction;
	DiagFunction_206:DiagFunction;
	DiagFunction_207:DiagFunction;
	DiagFunction_208:DiagFunction;
	
	DiagFunction_300:DiagFunction;
	DiagFunction_301:DiagFunction;
	DiagFunction_302:DiagFunction;
	DiagFunction_303:DiagFunction;
	DiagFunction_304:DiagFunction;
	DiagFunction_305:DiagFunction;
	DiagFunction_306:DiagFunction;
	DiagFunction_307:DiagFunction;
	DiagFunction_308:DiagFunction;
	
	DiagFunction_400:DiagFunction;
	DiagFunction_401:DiagFunction;
	DiagFunction_402:DiagFunction;
	DiagFunction_403:DiagFunction;
	DiagFunction_404:DiagFunction;
	DiagFunction_405:DiagFunction;
	DiagFunction_406:DiagFunction;
	DiagFunction_407:DiagFunction;
	DiagFunction_408:DiagFunction;
	
	DiagFunction_500:DiagFunction;
	DiagFunction_501:DiagFunction;
	DiagFunction_502:DiagFunction;
	DiagFunction_503:DiagFunction;
	DiagFunction_504:DiagFunction;
	DiagFunction_505:DiagFunction;
	DiagFunction_506:DiagFunction;
	DiagFunction_507:DiagFunction;
	DiagFunction_508:DiagFunction;	
	DiagFunction_Group0:DiagFunction;
	DiagFunction_Group1:DiagFunction;
	DiagFunction_Group2:DiagFunction;
	DiagFunction_Group3:DiagFunction;
	DiagFunction_Group4:DiagFunction;
	DiagFunction_Group5:DiagFunction;
	
	MinCurrent: UINT:=0;
	MaxCurrent: UINT:=2500;
	Time_: UINT:=1000;
	vagroup_1: BOOL:=TRUE;
	reset1: BOOL;
	
	ChangeVOL_A27: ifmConfigSwThreshold.ConfigSwThreshold;
	ChangeVOL_A28: ifmConfigSwThreshold.ConfigSwThreshold;
	ChangeVOL_A44: ifmConfigSwThreshold.ConfigSwThreshold;
	ChangeVOL_A45: ifmConfigSwThreshold.ConfigSwThreshold;


END_VAR

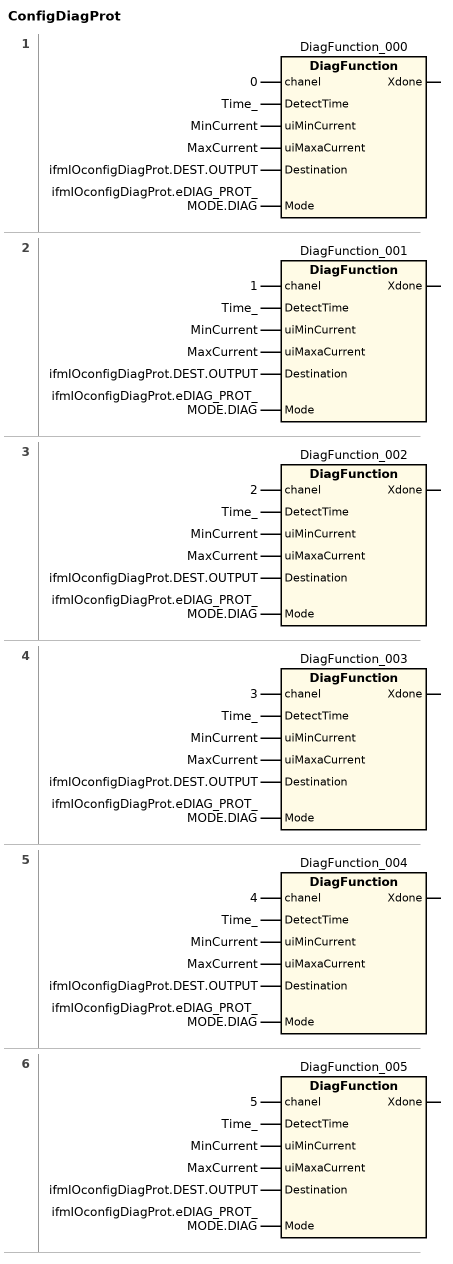
// NETWORK 1
DiagFunction_000(
    chanel := 0,
    DetectTime := Time_,
    uiMinCurrent := MinCurrent,
    uiMaxaCurrent := MaxCurrent,
    Destination := ifmIOconfigDiagProt.DEST.OUTPUT,
    Mode := ifmIOconfigDiagProt.eDIAG_PROT_MODE.DIAG); // DiagFunction

// NETWORK 2
DiagFunction_001(
    chanel := 1,
    DetectTime := Time_,
    uiMinCurrent := MinCurrent,
    uiMaxaCurrent := MaxCurrent,
    Destination := ifmIOconfigDiagProt.DEST.OUTPUT,
    Mode := ifmIOconfigDiagProt.eDIAG_PROT_MODE.DIAG); // DiagFunction

// NETWORK 3
DiagFunction_002(
    chanel := 2,
    DetectTime := Time_,
    uiMinCurrent := MinCurrent,
    uiMaxaCurrent := MaxCurrent,
    Destination := ifmIOconfigDiagProt.DEST.OUTPUT,
    Mode := ifmIOconfigDiagProt.eDIAG_PROT_MODE.DIAG); // DiagFunction

// NETWORK 4
DiagFunction_003(
    chanel := 3,
    DetectTime := Time_,
    uiMinCurrent := MinCurrent,
    uiMaxaCurrent := MaxCurrent,
    Destination := ifmIOconfigDiagProt.DEST.OUTPUT,
    Mode := ifmIOconfigDiagProt.eDIAG_PROT_MODE.DIAG); // DiagFunction

// NETWORK 5
DiagFunction_004(
    chanel := 4,
    DetectTime := Time_,
    uiMinCurrent := MinCurrent,
    uiMaxaCurrent := MaxCurrent,
    Destination := ifmIOconfigDiagProt.DEST.OUTPUT,
    Mode := ifmIOconfigDiagProt.eDIAG_PROT_MODE.DIAG); // DiagFunction

// NETWORK 6
DiagFunction_005(
    chanel := 5,
    DetectTime := Time_,
    uiMinCurrent := MinCurrent,
    uiMaxaCurrent := MaxCurrent,
    Destination := ifmIOconfigDiagProt.DEST.OUTPUT,
    Mode := ifmIOconfigDiagProt.eDIAG_PROT_MODE.DIAG); // DiagFunction

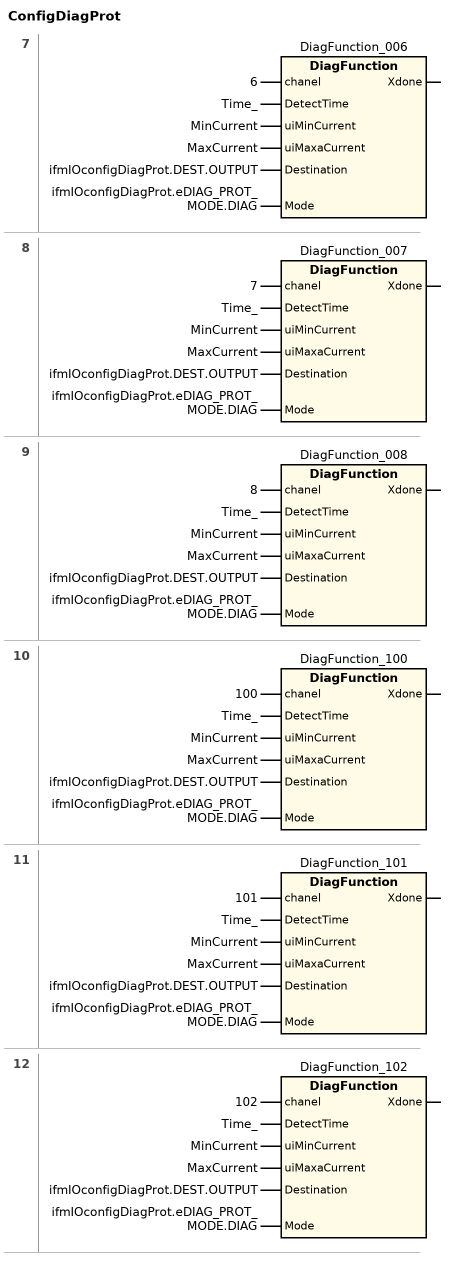
// NETWORK 7
DiagFunction_006(
    chanel := 6,
    DetectTime := Time_,
    uiMinCurrent := MinCurrent,
    uiMaxaCurrent := MaxCurrent,
    Destination := ifmIOconfigDiagProt.DEST.OUTPUT,
    Mode := ifmIOconfigDiagProt.eDIAG_PROT_MODE.DIAG); // DiagFunction

// NETWORK 8
DiagFunction_007(
    chanel := 7,
    DetectTime := Time_,
    uiMinCurrent := MinCurrent,
    uiMaxaCurrent := MaxCurrent,
    Destination := ifmIOconfigDiagProt.DEST.OUTPUT,
    Mode := ifmIOconfigDiagProt.eDIAG_PROT_MODE.DIAG); // DiagFunction

// NETWORK 9
DiagFunction_008(
    chanel := 8,
    DetectTime := Time_,
    uiMinCurrent := MinCurrent,
    uiMaxaCurrent := MaxCurrent,
    Destination := ifmIOconfigDiagProt.DEST.OUTPUT,
    Mode := ifmIOconfigDiagProt.eDIAG_PROT_MODE.DIAG); // DiagFunction

// NETWORK 10
DiagFunction_100(
    chanel := 100,
    DetectTime := Time_,
    uiMinCurrent := MinCurrent,
    uiMaxaCurrent := MaxCurrent,
    Destination := ifmIOconfigDiagProt.DEST.OUTPUT,
    Mode := ifmIOconfigDiagProt.eDIAG_PROT_MODE.DIAG); // DiagFunction

// NETWORK 11
DiagFunction_101(
    chanel := 101,
    DetectTime := Time_,
    uiMinCurrent := MinCurrent,
    uiMaxaCurrent := MaxCurrent,
    Destination := ifmIOconfigDiagProt.DEST.OUTPUT,
    Mode := ifmIOconfigDiagProt.eDIAG_PROT_MODE.DIAG); // DiagFunction

// NETWORK 12
DiagFunction_102(
    chanel := 102,
    DetectTime := Time_,
    uiMinCurrent := MinCurrent,
    uiMaxaCurrent := MaxCurrent,
    Destination := ifmIOconfigDiagProt.DEST.OUTPUT,
    Mode := ifmIOconfigDiagProt.eDIAG_PROT_MODE.DIAG); // DiagFunction

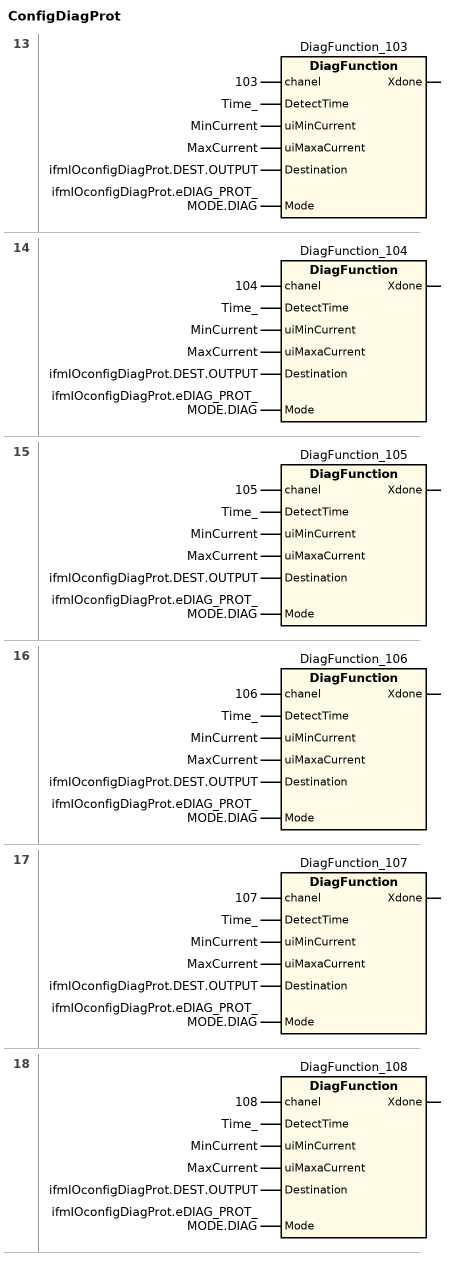
// NETWORK 13
DiagFunction_103(
    chanel := 103,
    DetectTime := Time_,
    uiMinCurrent := MinCurrent,
    uiMaxaCurrent := MaxCurrent,
    Destination := ifmIOconfigDiagProt.DEST.OUTPUT,
    Mode := ifmIOconfigDiagProt.eDIAG_PROT_MODE.DIAG); // DiagFunction

// NETWORK 14
DiagFunction_104(
    chanel := 104,
    DetectTime := Time_,
    uiMinCurrent := MinCurrent,
    uiMaxaCurrent := MaxCurrent,
    Destination := ifmIOconfigDiagProt.DEST.OUTPUT,
    Mode := ifmIOconfigDiagProt.eDIAG_PROT_MODE.DIAG); // DiagFunction

// NETWORK 15
DiagFunction_105(
    chanel := 105,
    DetectTime := Time_,
    uiMinCurrent := MinCurrent,
    uiMaxaCurrent := MaxCurrent,
    Destination := ifmIOconfigDiagProt.DEST.OUTPUT,
    Mode := ifmIOconfigDiagProt.eDIAG_PROT_MODE.DIAG); // DiagFunction

// NETWORK 16
DiagFunction_106(
    chanel := 106,
    DetectTime := Time_,
    uiMinCurrent := MinCurrent,
    uiMaxaCurrent := MaxCurrent,
    Destination := ifmIOconfigDiagProt.DEST.OUTPUT,
    Mode := ifmIOconfigDiagProt.eDIAG_PROT_MODE.DIAG); // DiagFunction

// NETWORK 17
DiagFunction_107(
    chanel := 107,
    DetectTime := Time_,
    uiMinCurrent := MinCurrent,
    uiMaxaCurrent := MaxCurrent,
    Destination := ifmIOconfigDiagProt.DEST.OUTPUT,
    Mode := ifmIOconfigDiagProt.eDIAG_PROT_MODE.DIAG); // DiagFunction

// NETWORK 18
DiagFunction_108(
    chanel := 108,
    DetectTime := Time_,
    uiMinCurrent := MinCurrent,
    uiMaxaCurrent := MaxCurrent,
    Destination := ifmIOconfigDiagProt.DEST.OUTPUT,
    Mode := ifmIOconfigDiagProt.eDIAG_PROT_MODE.DIAG); // DiagFunction

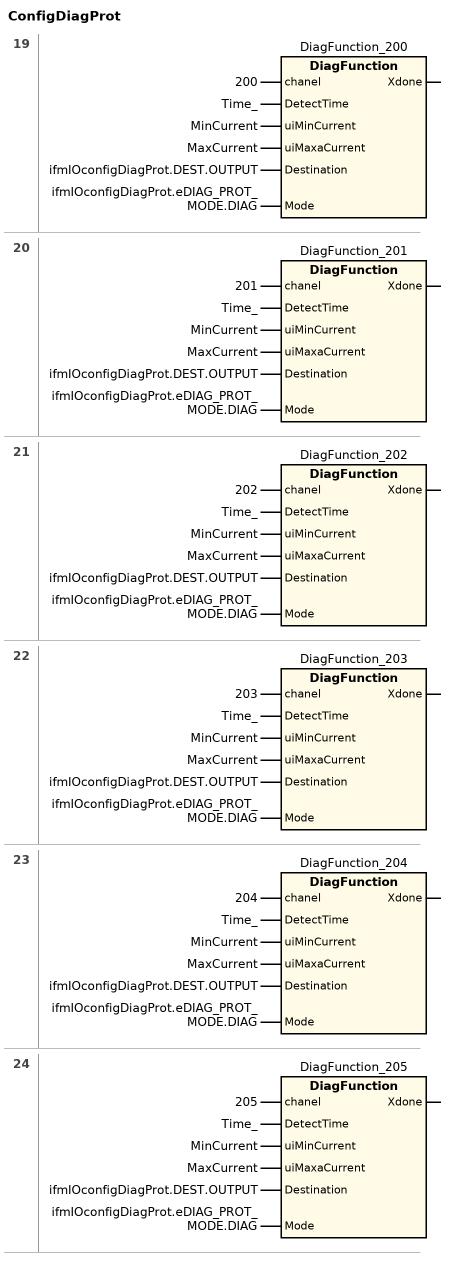
// NETWORK 19
DiagFunction_200(
    chanel := 200,
    DetectTime := Time_,
    uiMinCurrent := MinCurrent,
    uiMaxaCurrent := MaxCurrent,
    Destination := ifmIOconfigDiagProt.DEST.OUTPUT,
    Mode := ifmIOconfigDiagProt.eDIAG_PROT_MODE.DIAG); // DiagFunction

// NETWORK 20
DiagFunction_201(
    chanel := 201,
    DetectTime := Time_,
    uiMinCurrent := MinCurrent,
    uiMaxaCurrent := MaxCurrent,
    Destination := ifmIOconfigDiagProt.DEST.OUTPUT,
    Mode := ifmIOconfigDiagProt.eDIAG_PROT_MODE.DIAG); // DiagFunction

// NETWORK 21
DiagFunction_202(
    chanel := 202,
    DetectTime := Time_,
    uiMinCurrent := MinCurrent,
    uiMaxaCurrent := MaxCurrent,
    Destination := ifmIOconfigDiagProt.DEST.OUTPUT,
    Mode := ifmIOconfigDiagProt.eDIAG_PROT_MODE.DIAG); // DiagFunction

// NETWORK 22
DiagFunction_203(
    chanel := 203,
    DetectTime := Time_,
    uiMinCurrent := MinCurrent,
    uiMaxaCurrent := MaxCurrent,
    Destination := ifmIOconfigDiagProt.DEST.OUTPUT,
    Mode := ifmIOconfigDiagProt.eDIAG_PROT_MODE.DIAG); // DiagFunction

// NETWORK 23
DiagFunction_204(
    chanel := 204,
    DetectTime := Time_,
    uiMinCurrent := MinCurrent,
    uiMaxaCurrent := MaxCurrent,
    Destination := ifmIOconfigDiagProt.DEST.OUTPUT,
    Mode := ifmIOconfigDiagProt.eDIAG_PROT_MODE.DIAG); // DiagFunction

// NETWORK 24
DiagFunction_205(
    chanel := 205,
    DetectTime := Time_,
    uiMinCurrent := MinCurrent,
    uiMaxaCurrent := MaxCurrent,
    Destination := ifmIOconfigDiagProt.DEST.OUTPUT,
    Mode := ifmIOconfigDiagProt.eDIAG_PROT_MODE.DIAG); // DiagFunction

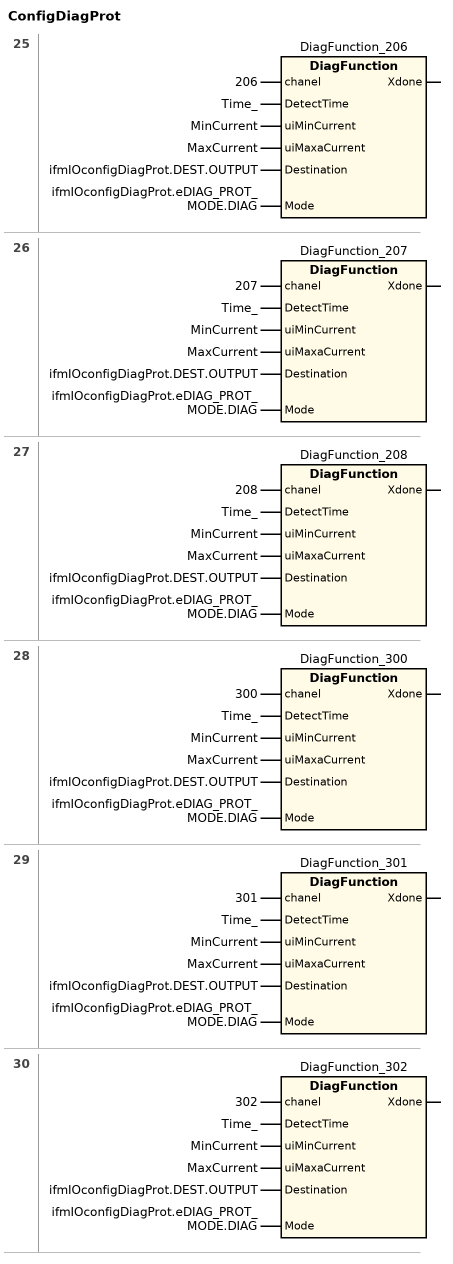
// NETWORK 25
DiagFunction_206(
    chanel := 206,
    DetectTime := Time_,
    uiMinCurrent := MinCurrent,
    uiMaxaCurrent := MaxCurrent,
    Destination := ifmIOconfigDiagProt.DEST.OUTPUT,
    Mode := ifmIOconfigDiagProt.eDIAG_PROT_MODE.DIAG); // DiagFunction

// NETWORK 26
DiagFunction_207(
    chanel := 207,
    DetectTime := Time_,
    uiMinCurrent := MinCurrent,
    uiMaxaCurrent := MaxCurrent,
    Destination := ifmIOconfigDiagProt.DEST.OUTPUT,
    Mode := ifmIOconfigDiagProt.eDIAG_PROT_MODE.DIAG); // DiagFunction

// NETWORK 27
DiagFunction_208(
    chanel := 208,
    DetectTime := Time_,
    uiMinCurrent := MinCurrent,
    uiMaxaCurrent := MaxCurrent,
    Destination := ifmIOconfigDiagProt.DEST.OUTPUT,
    Mode := ifmIOconfigDiagProt.eDIAG_PROT_MODE.DIAG); // DiagFunction

// NETWORK 28
DiagFunction_300(
    chanel := 300,
    DetectTime := Time_,
    uiMinCurrent := MinCurrent,
    uiMaxaCurrent := MaxCurrent,
    Destination := ifmIOconfigDiagProt.DEST.OUTPUT,
    Mode := ifmIOconfigDiagProt.eDIAG_PROT_MODE.DIAG); // DiagFunction

// NETWORK 29
DiagFunction_301(
    chanel := 301,
    DetectTime := Time_,
    uiMinCurrent := MinCurrent,
    uiMaxaCurrent := MaxCurrent,
    Destination := ifmIOconfigDiagProt.DEST.OUTPUT,
    Mode := ifmIOconfigDiagProt.eDIAG_PROT_MODE.DIAG); // DiagFunction

// NETWORK 30
DiagFunction_302(
    chanel := 302,
    DetectTime := Time_,
    uiMinCurrent := MinCurrent,
    uiMaxaCurrent := MaxCurrent,
    Destination := ifmIOconfigDiagProt.DEST.OUTPUT,
    Mode := ifmIOconfigDiagProt.eDIAG_PROT_MODE.DIAG); // DiagFunction

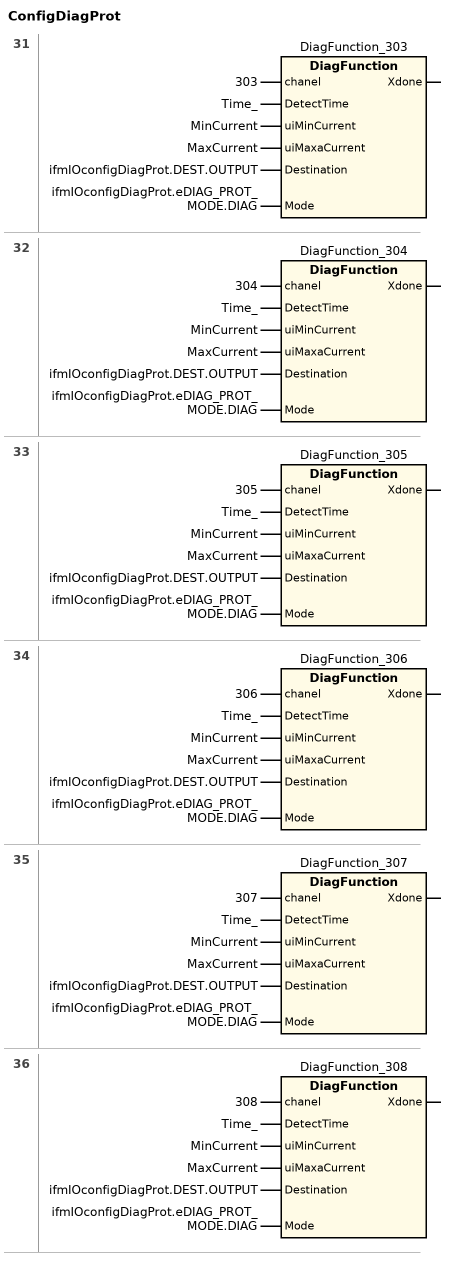
// NETWORK 31
DiagFunction_303(
    chanel := 303,
    DetectTime := Time_,
    uiMinCurrent := MinCurrent,
    uiMaxaCurrent := MaxCurrent,
    Destination := ifmIOconfigDiagProt.DEST.OUTPUT,
    Mode := ifmIOconfigDiagProt.eDIAG_PROT_MODE.DIAG); // DiagFunction

// NETWORK 32
DiagFunction_304(
    chanel := 304,
    DetectTime := Time_,
    uiMinCurrent := MinCurrent,
    uiMaxaCurrent := MaxCurrent,
    Destination := ifmIOconfigDiagProt.DEST.OUTPUT,
    Mode := ifmIOconfigDiagProt.eDIAG_PROT_MODE.DIAG); // DiagFunction

// NETWORK 33
DiagFunction_305(
    chanel := 305,
    DetectTime := Time_,
    uiMinCurrent := MinCurrent,
    uiMaxaCurrent := MaxCurrent,
    Destination := ifmIOconfigDiagProt.DEST.OUTPUT,
    Mode := ifmIOconfigDiagProt.eDIAG_PROT_MODE.DIAG); // DiagFunction

// NETWORK 34
DiagFunction_306(
    chanel := 306,
    DetectTime := Time_,
    uiMinCurrent := MinCurrent,
    uiMaxaCurrent := MaxCurrent,
    Destination := ifmIOconfigDiagProt.DEST.OUTPUT,
    Mode := ifmIOconfigDiagProt.eDIAG_PROT_MODE.DIAG); // DiagFunction

// NETWORK 35
DiagFunction_307(
    chanel := 307,
    DetectTime := Time_,
    uiMinCurrent := MinCurrent,
    uiMaxaCurrent := MaxCurrent,
    Destination := ifmIOconfigDiagProt.DEST.OUTPUT,
    Mode := ifmIOconfigDiagProt.eDIAG_PROT_MODE.DIAG); // DiagFunction

// NETWORK 36
DiagFunction_308(
    chanel := 308,
    DetectTime := Time_,
    uiMinCurrent := MinCurrent,
    uiMaxaCurrent := MaxCurrent,
    Destination := ifmIOconfigDiagProt.DEST.OUTPUT,
    Mode := ifmIOconfigDiagProt.eDIAG_PROT_MODE.DIAG); // DiagFunction

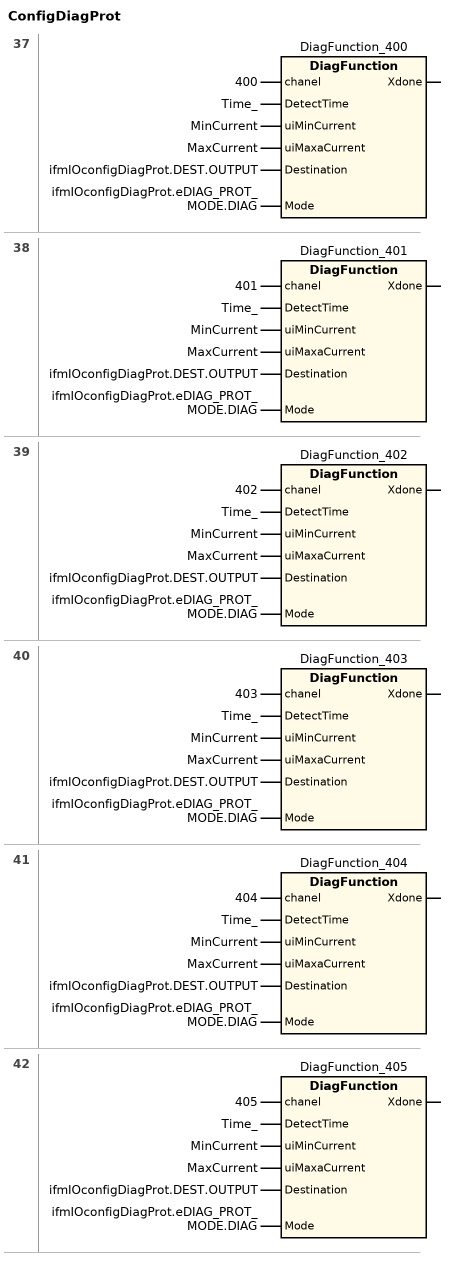
// NETWORK 37
DiagFunction_400(
    chanel := 400,
    DetectTime := Time_,
    uiMinCurrent := MinCurrent,
    uiMaxaCurrent := MaxCurrent,
    Destination := ifmIOconfigDiagProt.DEST.OUTPUT,
    Mode := ifmIOconfigDiagProt.eDIAG_PROT_MODE.DIAG); // DiagFunction

// NETWORK 38
DiagFunction_401(
    chanel := 401,
    DetectTime := Time_,
    uiMinCurrent := MinCurrent,
    uiMaxaCurrent := MaxCurrent,
    Destination := ifmIOconfigDiagProt.DEST.OUTPUT,
    Mode := ifmIOconfigDiagProt.eDIAG_PROT_MODE.DIAG); // DiagFunction

// NETWORK 39
DiagFunction_402(
    chanel := 402,
    DetectTime := Time_,
    uiMinCurrent := MinCurrent,
    uiMaxaCurrent := MaxCurrent,
    Destination := ifmIOconfigDiagProt.DEST.OUTPUT,
    Mode := ifmIOconfigDiagProt.eDIAG_PROT_MODE.DIAG); // DiagFunction

// NETWORK 40
DiagFunction_403(
    chanel := 403,
    DetectTime := Time_,
    uiMinCurrent := MinCurrent,
    uiMaxaCurrent := MaxCurrent,
    Destination := ifmIOconfigDiagProt.DEST.OUTPUT,
    Mode := ifmIOconfigDiagProt.eDIAG_PROT_MODE.DIAG); // DiagFunction

// NETWORK 41
DiagFunction_404(
    chanel := 404,
    DetectTime := Time_,
    uiMinCurrent := MinCurrent,
    uiMaxaCurrent := MaxCurrent,
    Destination := ifmIOconfigDiagProt.DEST.OUTPUT,
    Mode := ifmIOconfigDiagProt.eDIAG_PROT_MODE.DIAG); // DiagFunction

// NETWORK 42
DiagFunction_405(
    chanel := 405,
    DetectTime := Time_,
    uiMinCurrent := MinCurrent,
    uiMaxaCurrent := MaxCurrent,
    Destination := ifmIOconfigDiagProt.DEST.OUTPUT,
    Mode := ifmIOconfigDiagProt.eDIAG_PROT_MODE.DIAG); // DiagFunction

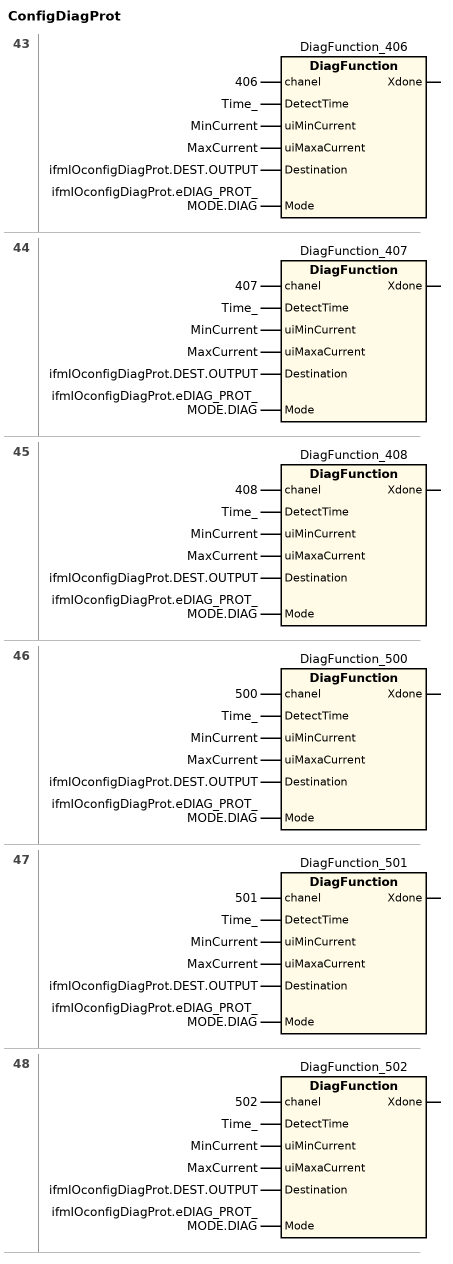
// NETWORK 43
DiagFunction_406(
    chanel := 406,
    DetectTime := Time_,
    uiMinCurrent := MinCurrent,
    uiMaxaCurrent := MaxCurrent,
    Destination := ifmIOconfigDiagProt.DEST.OUTPUT,
    Mode := ifmIOconfigDiagProt.eDIAG_PROT_MODE.DIAG); // DiagFunction

// NETWORK 44
DiagFunction_407(
    chanel := 407,
    DetectTime := Time_,
    uiMinCurrent := MinCurrent,
    uiMaxaCurrent := MaxCurrent,
    Destination := ifmIOconfigDiagProt.DEST.OUTPUT,
    Mode := ifmIOconfigDiagProt.eDIAG_PROT_MODE.DIAG); // DiagFunction

// NETWORK 45
DiagFunction_408(
    chanel := 408,
    DetectTime := Time_,
    uiMinCurrent := MinCurrent,
    uiMaxaCurrent := MaxCurrent,
    Destination := ifmIOconfigDiagProt.DEST.OUTPUT,
    Mode := ifmIOconfigDiagProt.eDIAG_PROT_MODE.DIAG); // DiagFunction

// NETWORK 46
DiagFunction_500(
    chanel := 500,
    DetectTime := Time_,
    uiMinCurrent := MinCurrent,
    uiMaxaCurrent := MaxCurrent,
    Destination := ifmIOconfigDiagProt.DEST.OUTPUT,
    Mode := ifmIOconfigDiagProt.eDIAG_PROT_MODE.DIAG); // DiagFunction

// NETWORK 47
DiagFunction_501(
    chanel := 501,
    DetectTime := Time_,
    uiMinCurrent := MinCurrent,
    uiMaxaCurrent := MaxCurrent,
    Destination := ifmIOconfigDiagProt.DEST.OUTPUT,
    Mode := ifmIOconfigDiagProt.eDIAG_PROT_MODE.DIAG); // DiagFunction

// NETWORK 48
DiagFunction_502(
    chanel := 502,
    DetectTime := Time_,
    uiMinCurrent := MinCurrent,
    uiMaxaCurrent := MaxCurrent,
    Destination := ifmIOconfigDiagProt.DEST.OUTPUT,
    Mode := ifmIOconfigDiagProt.eDIAG_PROT_MODE.DIAG); // DiagFunction

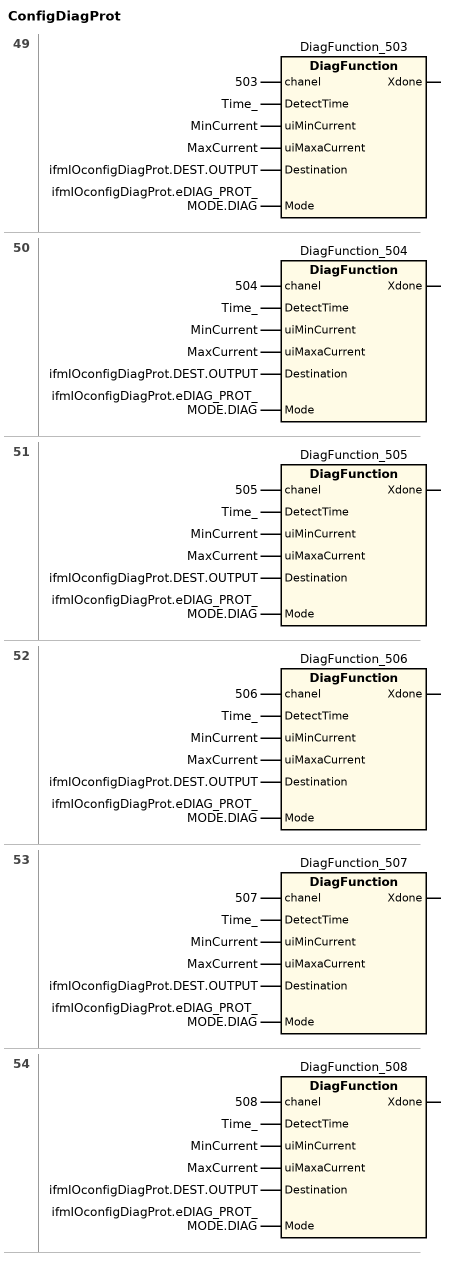
// NETWORK 49
DiagFunction_503(
    chanel := 503,
    DetectTime := Time_,
    uiMinCurrent := MinCurrent,
    uiMaxaCurrent := MaxCurrent,
    Destination := ifmIOconfigDiagProt.DEST.OUTPUT,
    Mode := ifmIOconfigDiagProt.eDIAG_PROT_MODE.DIAG); // DiagFunction

// NETWORK 50
DiagFunction_504(
    chanel := 504,
    DetectTime := Time_,
    uiMinCurrent := MinCurrent,
    uiMaxaCurrent := MaxCurrent,
    Destination := ifmIOconfigDiagProt.DEST.OUTPUT,
    Mode := ifmIOconfigDiagProt.eDIAG_PROT_MODE.DIAG); // DiagFunction

// NETWORK 51
DiagFunction_505(
    chanel := 505,
    DetectTime := Time_,
    uiMinCurrent := MinCurrent,
    uiMaxaCurrent := MaxCurrent,
    Destination := ifmIOconfigDiagProt.DEST.OUTPUT,
    Mode := ifmIOconfigDiagProt.eDIAG_PROT_MODE.DIAG); // DiagFunction

// NETWORK 52
DiagFunction_506(
    chanel := 506,
    DetectTime := Time_,
    uiMinCurrent := MinCurrent,
    uiMaxaCurrent := MaxCurrent,
    Destination := ifmIOconfigDiagProt.DEST.OUTPUT,
    Mode := ifmIOconfigDiagProt.eDIAG_PROT_MODE.DIAG); // DiagFunction

// NETWORK 53
DiagFunction_507(
    chanel := 507,
    DetectTime := Time_,
    uiMinCurrent := MinCurrent,
    uiMaxaCurrent := MaxCurrent,
    Destination := ifmIOconfigDiagProt.DEST.OUTPUT,
    Mode := ifmIOconfigDiagProt.eDIAG_PROT_MODE.DIAG); // DiagFunction

// NETWORK 54
DiagFunction_508(
    chanel := 508,
    DetectTime := Time_,
    uiMinCurrent := MinCurrent,
    uiMaxaCurrent := MaxCurrent,
    Destination := ifmIOconfigDiagProt.DEST.OUTPUT,
    Mode := ifmIOconfigDiagProt.eDIAG_PROT_MODE.DIAG); // DiagFunction

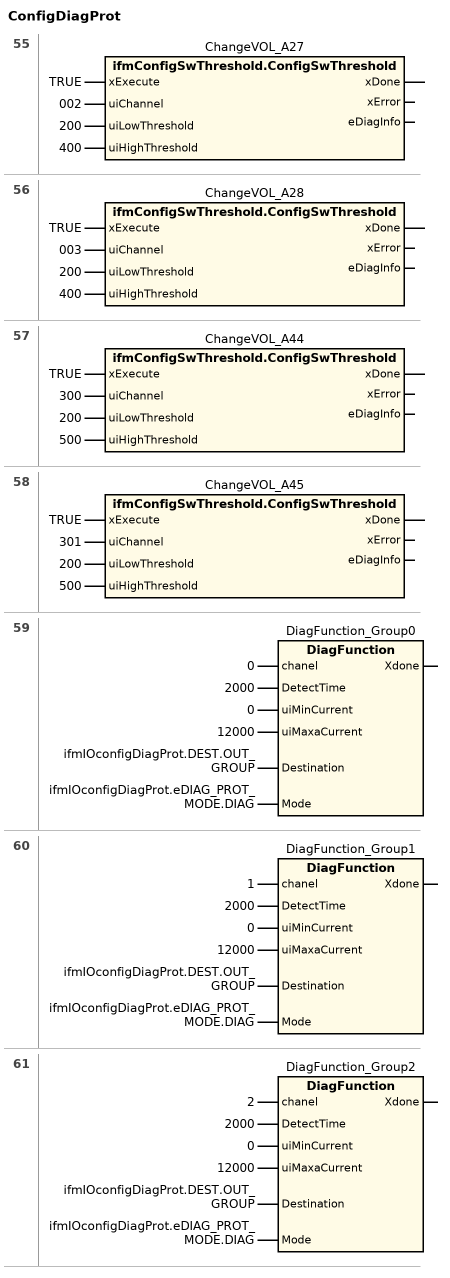
// NETWORK 55
ChangeVOL_A27(xExecute := TRUE, uiChannel := 002, uiLowThreshold := 200, uiHighThreshold := 400); // ifmConfigSwThreshold.ConfigSwThreshold

// NETWORK 56
ChangeVOL_A28(xExecute := TRUE, uiChannel := 003, uiLowThreshold := 200, uiHighThreshold := 400); // ifmConfigSwThreshold.ConfigSwThreshold

// NETWORK 57
ChangeVOL_A44(xExecute := TRUE, uiChannel := 300, uiLowThreshold := 200, uiHighThreshold := 500); // ifmConfigSwThreshold.ConfigSwThreshold

// NETWORK 58
ChangeVOL_A45(xExecute := TRUE, uiChannel := 301, uiLowThreshold := 200, uiHighThreshold := 500); // ifmConfigSwThreshold.ConfigSwThreshold

// NETWORK 59
DiagFunction_Group0(
    chanel := 0,
    DetectTime := 2000,
    uiMinCurrent := 0,
    uiMaxaCurrent := 12000,
    Destination := ifmIOconfigDiagProt.DEST.OUT_GROUP,
    Mode := ifmIOconfigDiagProt.eDIAG_PROT_MODE.DIAG); // DiagFunction

// NETWORK 60
DiagFunction_Group1(
    chanel := 1,
    DetectTime := 2000,
    uiMinCurrent := 0,
    uiMaxaCurrent := 12000,
    Destination := ifmIOconfigDiagProt.DEST.OUT_GROUP,
    Mode := ifmIOconfigDiagProt.eDIAG_PROT_MODE.DIAG); // DiagFunction

// NETWORK 61
DiagFunction_Group2(
    chanel := 2,
    DetectTime := 2000,
    uiMinCurrent := 0,
    uiMaxaCurrent := 12000,
    Destination := ifmIOconfigDiagProt.DEST.OUT_GROUP,
    Mode := ifmIOconfigDiagProt.eDIAG_PROT_MODE.DIAG); // DiagFunction

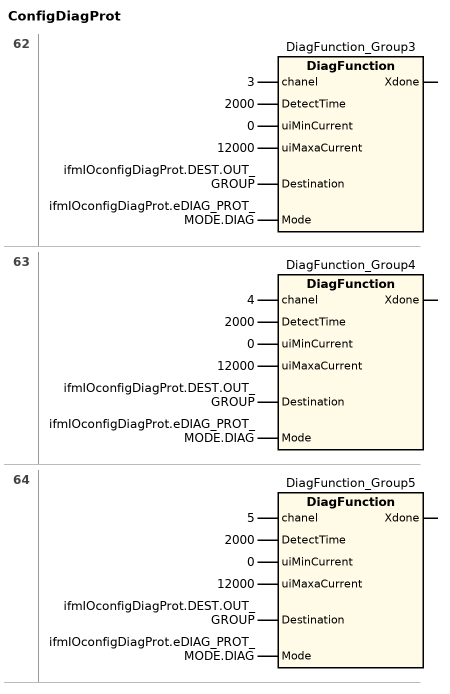
// NETWORK 62
DiagFunction_Group3(
    chanel := 3,
    DetectTime := 2000,
    uiMinCurrent := 0,
    uiMaxaCurrent := 12000,
    Destination := ifmIOconfigDiagProt.DEST.OUT_GROUP,
    Mode := ifmIOconfigDiagProt.eDIAG_PROT_MODE.DIAG); // DiagFunction

// NETWORK 63
DiagFunction_Group4(
    chanel := 4,
    DetectTime := 2000,
    uiMinCurrent := 0,
    uiMaxaCurrent := 12000,
    Destination := ifmIOconfigDiagProt.DEST.OUT_GROUP,
    Mode := ifmIOconfigDiagProt.eDIAG_PROT_MODE.DIAG); // DiagFunction

// NETWORK 64
DiagFunction_Group5(
    chanel := 5,
    DetectTime := 2000,
    uiMinCurrent := 0,
    uiMaxaCurrent := 12000,
    Destination := ifmIOconfigDiagProt.DEST.OUT_GROUP,
    Mode := ifmIOconfigDiagProt.eDIAG_PROT_MODE.DIAG); // DiagFunction

END_PROGRAM

// StandardPLC/Application/IO_CONFIG/DiagFunction
FUNCTION_BLOCK DiagFunction
VAR_INPUT
	chanel: UINT;
	DetectTime: UINT;
	uiMinCurrent: UINT;
	uiMaxaCurrent: UINT;
	Destination: ifmIOconfigDiagProt.DEST;
	Mode: ifmIOconfigDiagProt.eDIAG_PROT_MODE;
END_VAR
VAR_OUTPUT	
	Xdone: BOOL;
END_VAR
VAR
	ConfigDiagProt_0: ifmIOconfigDiagProt.ConfigDiagProt;
	init0: BOOL:=TRUE;
	ConfigDiagProt_1: ifmIOconfigDiagProt.ConfigDiagLevel;
	init1: BOOL:=true;
END_VAR

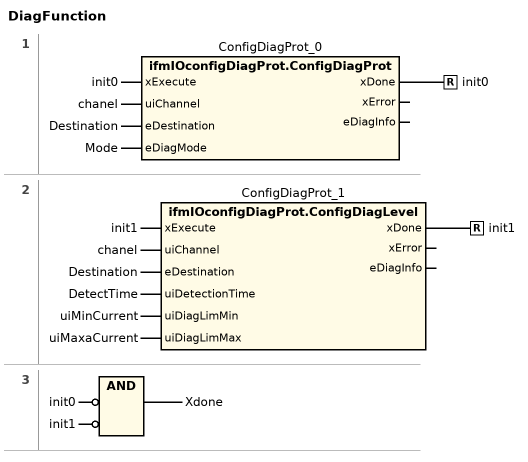
// NETWORK 1
ConfigDiagProt_0(xExecute := init0, uiChannel := chanel, eDestination := Destination, eDiagMode := Mode); // ifmIOconfigDiagProt.ConfigDiagProt
init0 R= ConfigDiagProt_0.xDone;

// NETWORK 2
ConfigDiagProt_1(
    xExecute := init1,
    uiChannel := chanel,
    eDestination := Destination,
    uiDetectionTime := DetectTime,
    uiDiagLimMin := uiMinCurrent,
    uiDiagLimMax := uiMaxaCurrent); // ifmIOconfigDiagProt.ConfigDiagLevel
init1 R= ConfigDiagProt_1.xDone;

// NETWORK 3
Xdone := NOT init0 AND NOT init1;

END_FUNCTION_BLOCK

